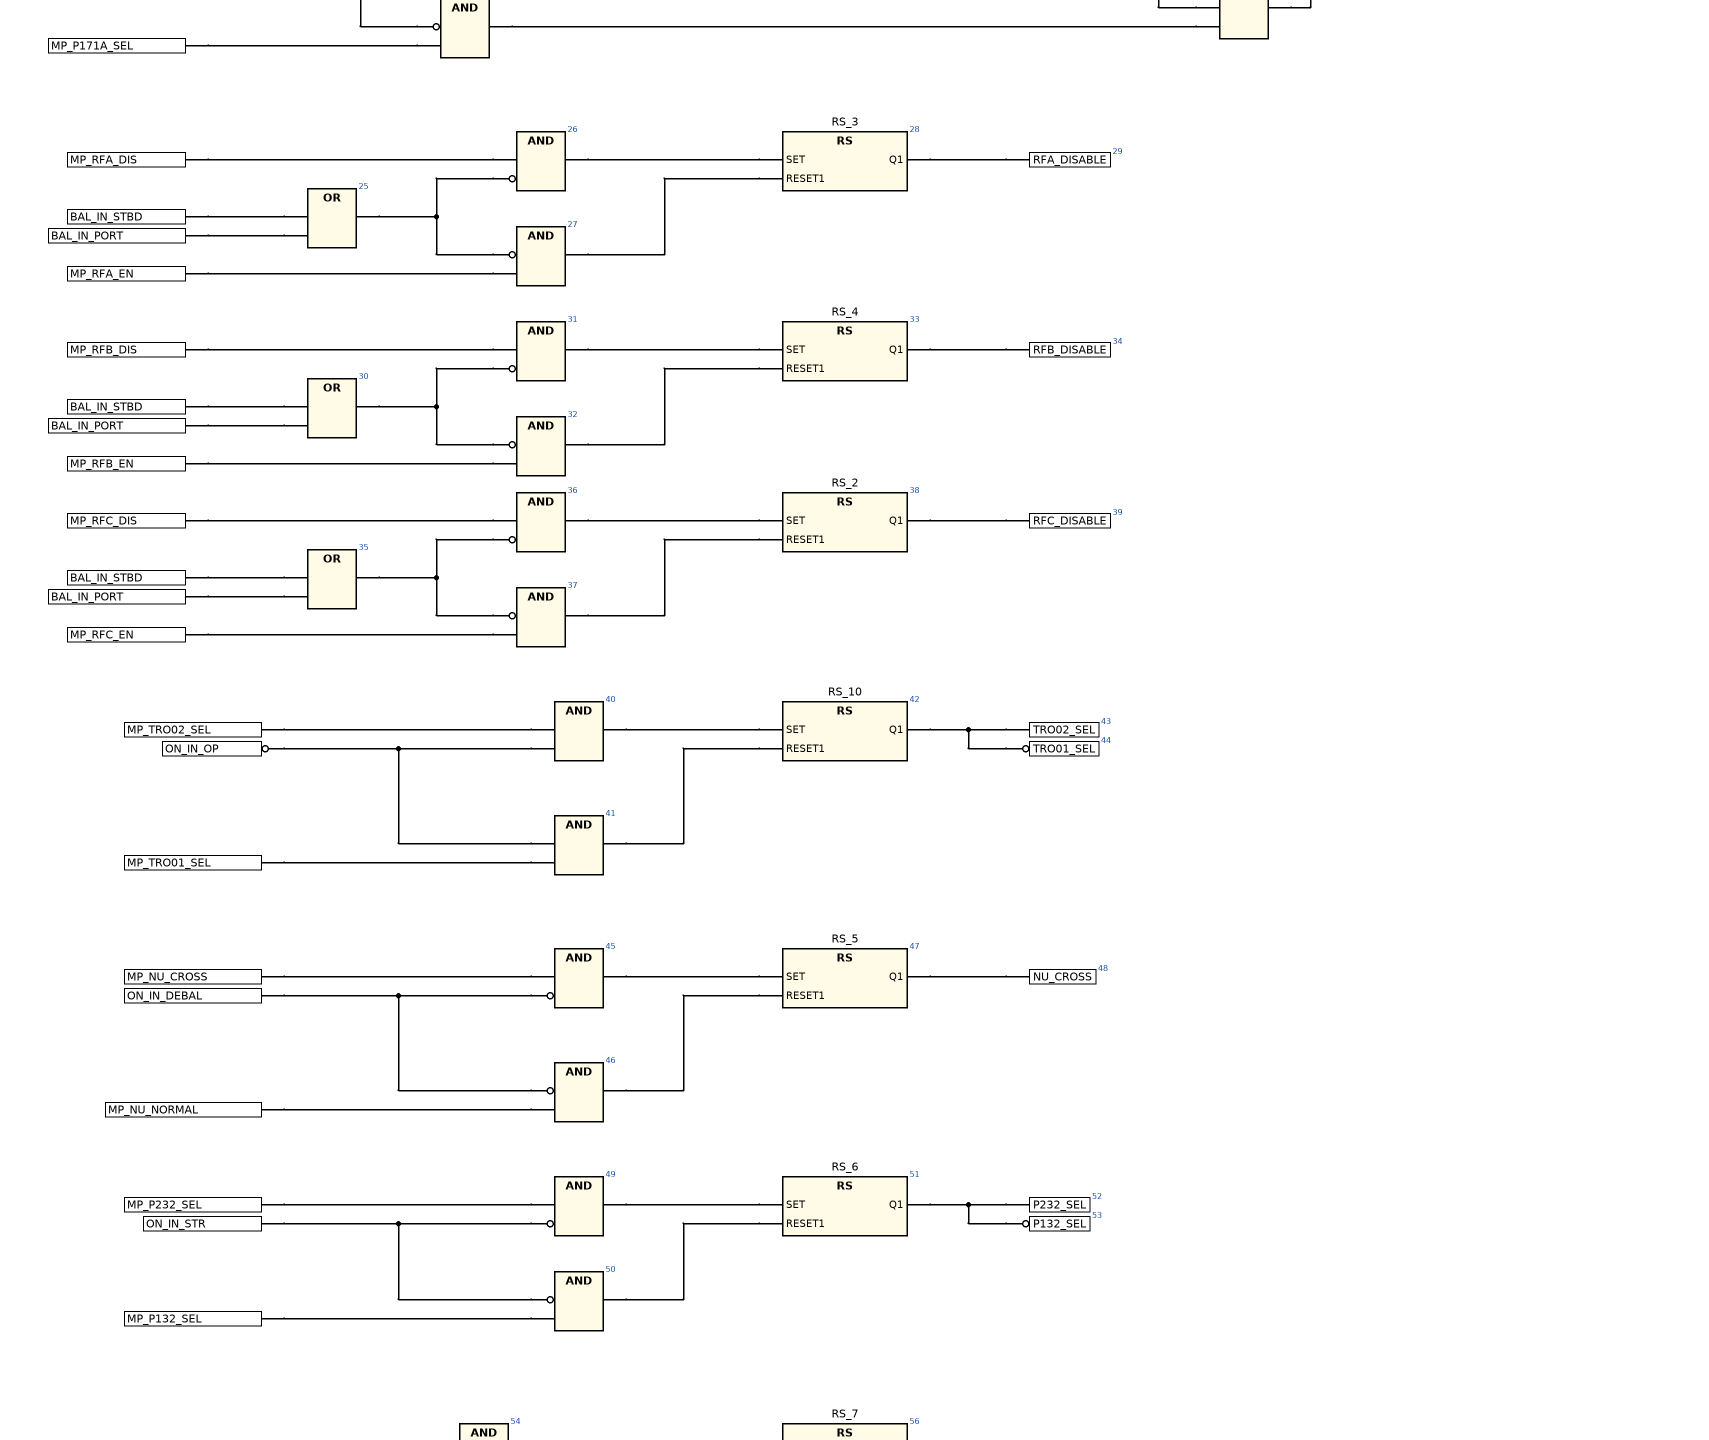
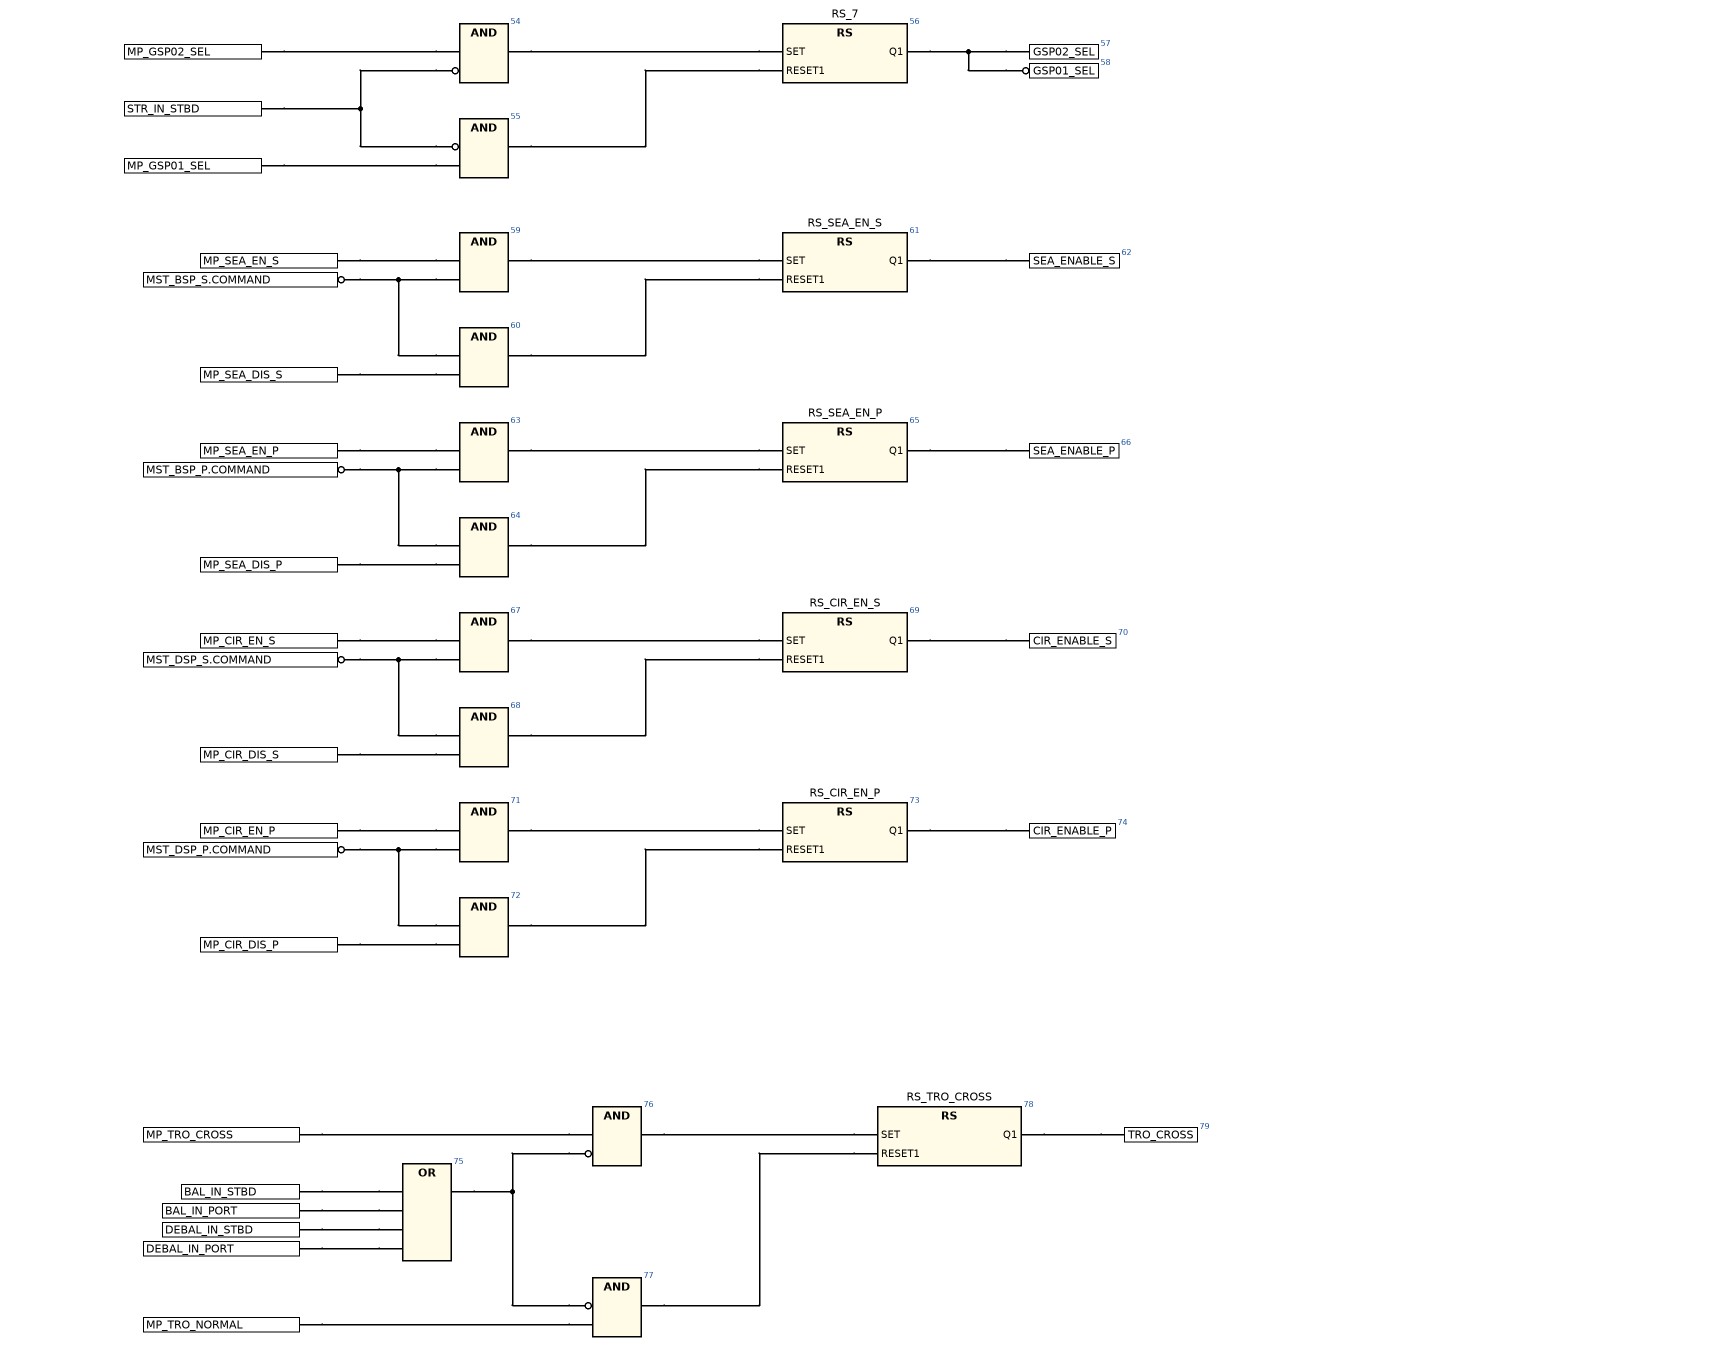
_w1 := ON_IN_BAL OR BLOWER_TIMER.BLR_GAS_SET.Q1;
RS_0(SET := MP_B117B_SEL AND NOT ON_IN_BAL OR B117A_SEL AND (B117A_STF OR XV1171A_OPF OR B_117A_F OR B_117A_OFF) AND _w1, RESET1 := NOT ON_IN_BAL AND MP_B117A_SEL OR _w1 AND B117B_SEL AND (B117B_STF OR XV1171B_OPF OR B_117B_F OR B_117B_OFF)); // RS
B117A_SEL := NOT RS_0.Q1;
B117B_SEL := RS_0.Q1;
_w2 := BAL_IN_STBD OR BAL_IN_PORT;
_w3 := BST_S_06.COMMAND OR BST_S_06.COMPLETE OR BST_P_06.COMMAND OR BST_P_06.COMPLETE;
RS_1(SET := MP_P171B_SEL AND NOT _w2 OR P171A_SEL AND (P171A_STF OR P_171A_OFF OR P_171A_F) AND _w3, RESET1 := _w3 AND P171B_SEL AND (P171B_STF OR P_171B_OFF OR P_171B_F) OR NOT _w2 AND MP_P171A_SEL); // RS
P171A_SEL := NOT RS_1.Q1;
P171B_SEL := RS_1.Q1;
_w4 := BAL_IN_STBD OR BAL_IN_PORT;
RS_3(SET := MP_RFA_DIS AND NOT _w4, RESET1 := NOT _w4 AND MP_RFA_EN); // RS
RFA_DISABLE := RS_3.Q1;
_w5 := BAL_IN_STBD OR BAL_IN_PORT;
RS_4(SET := MP_RFB_DIS AND NOT _w5, RESET1 := NOT _w5 AND MP_RFB_EN); // RS
RFB_DISABLE := RS_4.Q1;
_w6 := BAL_IN_STBD OR BAL_IN_PORT;
RS_2(SET := MP_RFC_DIS AND NOT _w6, RESET1 := NOT _w6 AND MP_RFC_EN); // RS
RFC_DISABLE := RS_2.Q1;
RS_10(SET := MP_TRO02_SEL AND NOT ON_IN_OP, RESET1 := NOT ON_IN_OP AND MP_TRO01_SEL); // RS
TRO02_SEL := RS_10.Q1;
TRO01_SEL := NOT RS_10.Q1;
RS_5(SET := MP_NU_CROSS AND NOT ON_IN_DEBAL, RESET1 := NOT ON_IN_DEBAL AND MP_NU_NORMAL); // RS
NU_CROSS := RS_5.Q1;
RS_6(SET := MP_P232_SEL AND NOT ON_IN_STR, RESET1 := NOT ON_IN_STR AND MP_P132_SEL); // RS
P232_SEL := RS_6.Q1;
P132_SEL := NOT RS_6.Q1;
RS_7(SET := MP_GSP02_SEL AND NOT STR_IN_STBD, RESET1 := NOT STR_IN_STBD AND MP_GSP01_SEL); // RS
GSP02_SEL := RS_7.Q1;
GSP01_SEL := NOT RS_7.Q1;
RS_SEA_EN_S(SET := MP_SEA_EN_S AND NOT MST_BSP_S.COMMAND, RESET1 := NOT MST_BSP_S.COMMAND AND MP_SEA_DIS_S); // RS
SEA_ENABLE_S := RS_SEA_EN_S.Q1;
RS_SEA_EN_P(SET := MP_SEA_EN_P AND NOT MST_BSP_P.COMMAND, RESET1 := NOT MST_BSP_P.COMMAND AND MP_SEA_DIS_P); // RS
SEA_ENABLE_P := RS_SEA_EN_P.Q1;
RS_CIR_EN_S(SET := MP_CIR_EN_S AND NOT MST_DSP_S.COMMAND, RESET1 := NOT MST_DSP_S.COMMAND AND MP_CIR_DIS_S); // RS
CIR_ENABLE_S := RS_CIR_EN_S.Q1;
RS_CIR_EN_P(SET := MP_CIR_EN_P AND NOT MST_DSP_P.COMMAND, RESET1 := NOT MST_DSP_P.COMMAND AND MP_CIR_DIS_P); // RS
CIR_ENABLE_P := RS_CIR_EN_P.Q1;
_w7 := BAL_IN_STBD OR BAL_IN_PORT OR DEBAL_IN_STBD OR DEBAL_IN_PORT;
RS_TRO_CROSS(SET := MP_TRO_CROSS AND NOT _w7, RESET1 := NOT _w7 AND MP_TRO_NORMAL); // RS
TRO_CROSS := RS_TRO_CROSS.Q1;

END_PROGRAM

// Device/Application/Logic/0.ETC/UTILITY
PROGRAM UTILITY
VAR
	INJECTION_SET: BWTS.INJECTION_SET;
	
		
	RS_BAL_ST_M : RS;
	TP_BAL_SP_M : TP;
	RS_DEBAL_ST_M : RS;
	TP_DEBAL_SP_M : TP;	
	RS_STRIP_ST : RS;
	TP_STRIP_SP : TP;
	
	RS_RFA_ST : RS;
	TP_RFA_SP : TP;
	RS_RFB_ST : RS;
	TP_RFB_SP : TP;
	RS_RFC_ST : RS;
	TP_RFC_SP : TP; 
	
	NA_PRE_SET_P132 : BWTS.NA_PRE_SET;
	NA_PRE_SET_P232 : BWTS.NA_PRE_SET;
		
	NA_CAPA_N1 : REAL := 31.2;
	NA_CAPA_N2 : REAL := 61.5;
	NA_CAPA_N3 : REAL := 129;
	NA_CAPA_N4 : REAL := 244.8;
END_VAR
VAR // added by the converter: edge detectors and wires of the graphical bodies
    _w1 : ANY;
END_VAR

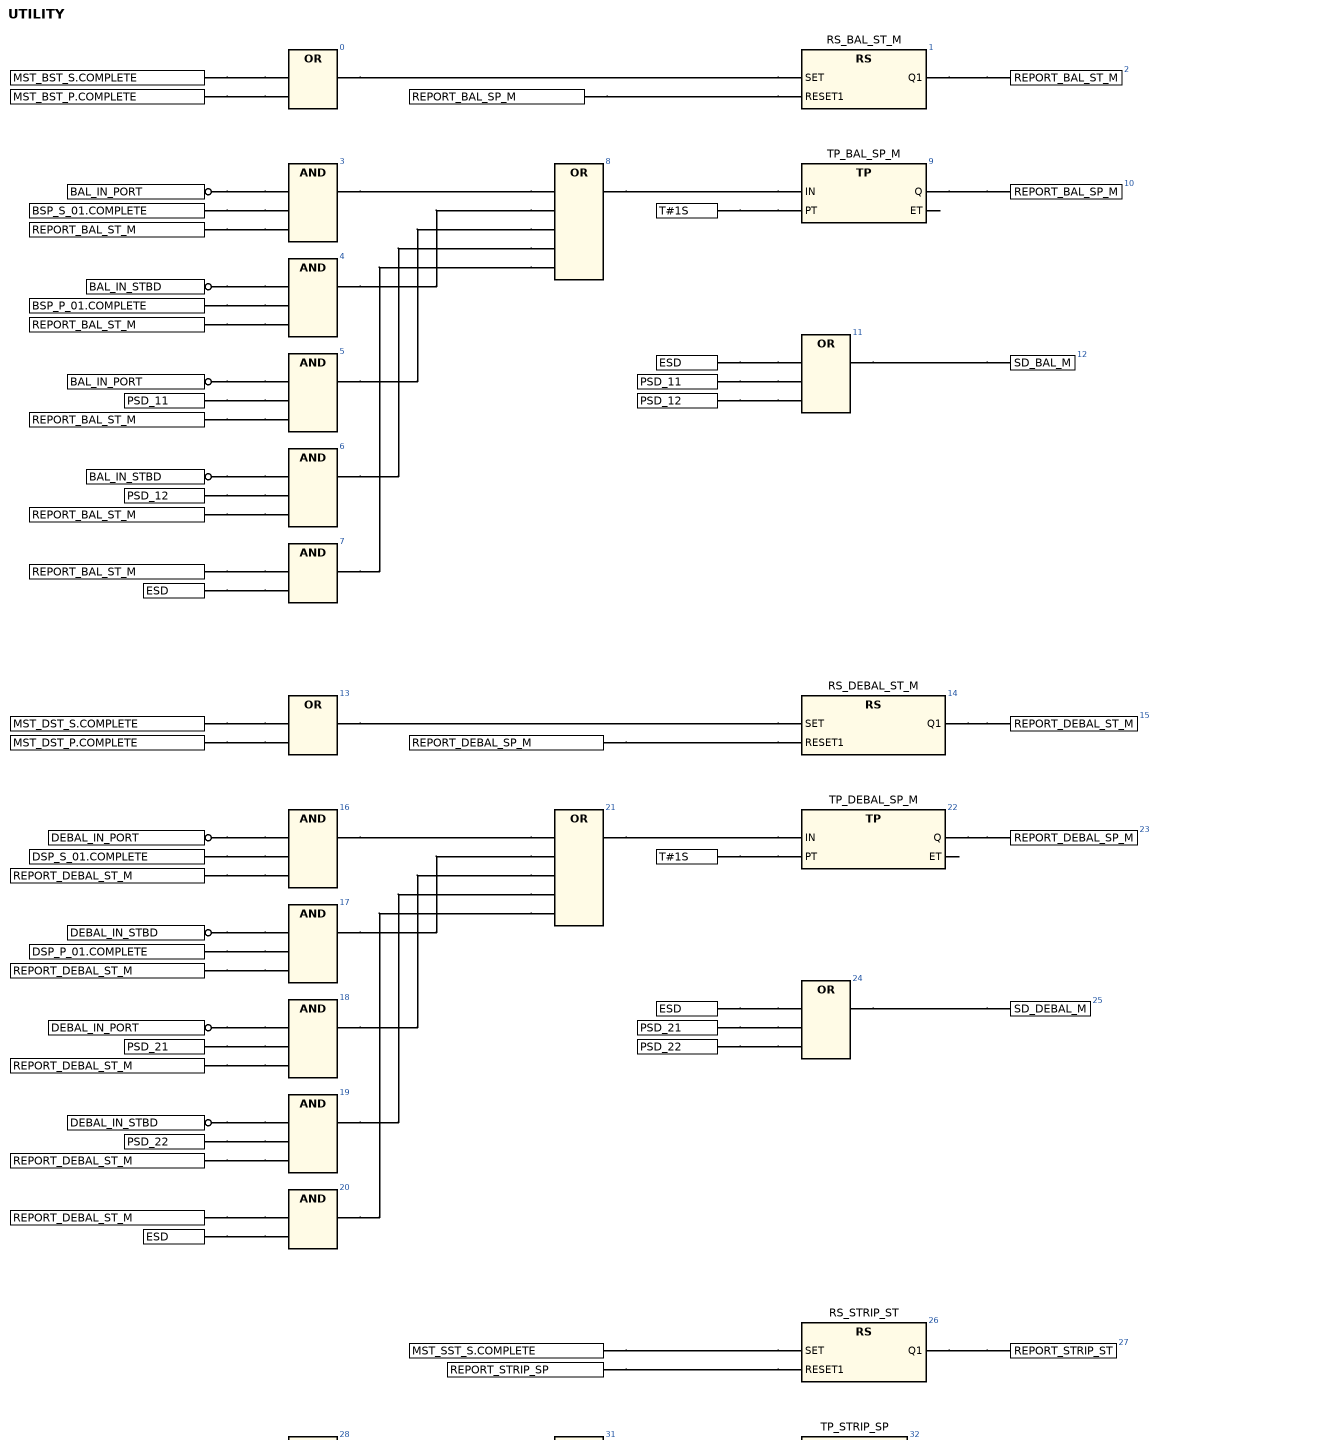
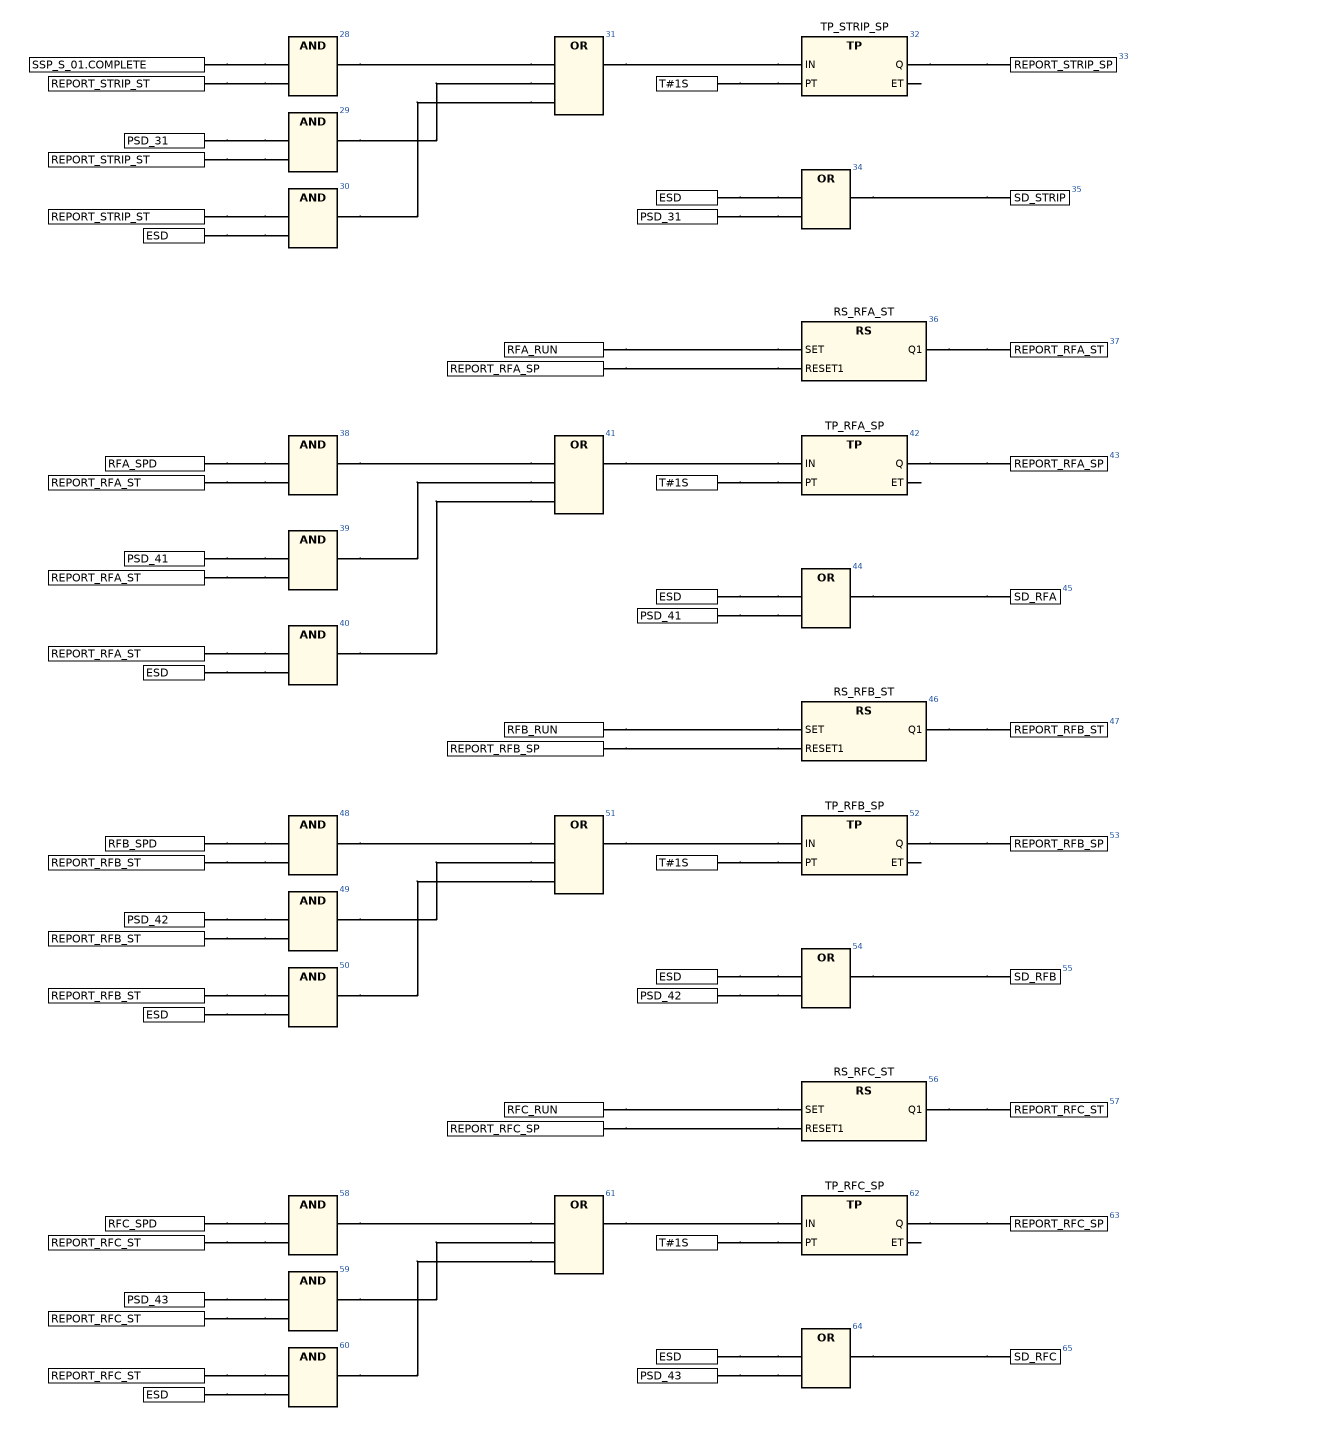
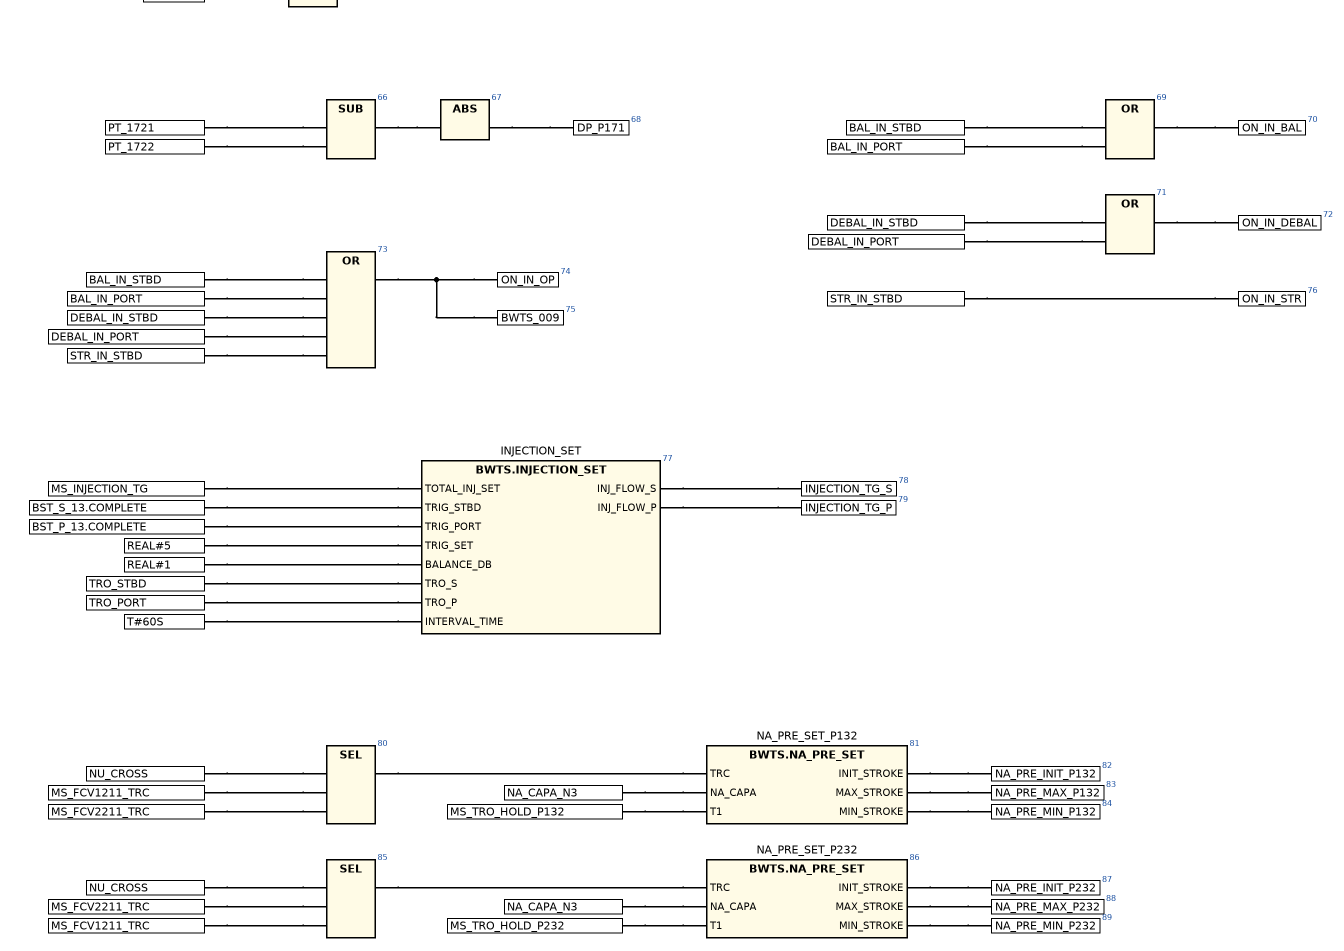
RS_BAL_ST_M(SET := MST_BST_S.COMPLETE OR MST_BST_P.COMPLETE, RESET1 := REPORT_BAL_SP_M); // RS
REPORT_BAL_ST_M := RS_BAL_ST_M.Q1;
TP_BAL_SP_M(IN := NOT BAL_IN_PORT AND BSP_S_01.COMPLETE AND REPORT_BAL_ST_M OR NOT BAL_IN_STBD AND BSP_P_01.COMPLETE AND REPORT_BAL_ST_M OR NOT BAL_IN_PORT AND PSD_11 AND REPORT_BAL_ST_M OR NOT BAL_IN_STBD AND PSD_12 AND REPORT_BAL_ST_M OR REPORT_BAL_ST_M AND ESD, PT := T#1S); // TP
REPORT_BAL_SP_M := TP_BAL_SP_M.Q;
SD_BAL_M := ESD OR PSD_11 OR PSD_12;
RS_DEBAL_ST_M(SET := MST_DST_S.COMPLETE OR MST_DST_P.COMPLETE, RESET1 := REPORT_DEBAL_SP_M); // RS
REPORT_DEBAL_ST_M := RS_DEBAL_ST_M.Q1;
TP_DEBAL_SP_M(IN := NOT DEBAL_IN_PORT AND DSP_S_01.COMPLETE AND REPORT_DEBAL_ST_M OR NOT DEBAL_IN_STBD AND DSP_P_01.COMPLETE AND REPORT_DEBAL_ST_M OR NOT DEBAL_IN_PORT AND PSD_21 AND REPORT_DEBAL_ST_M OR NOT DEBAL_IN_STBD AND PSD_22 AND REPORT_DEBAL_ST_M OR REPORT_DEBAL_ST_M AND ESD, PT := T#1S); // TP
REPORT_DEBAL_SP_M := TP_DEBAL_SP_M.Q;
SD_DEBAL_M := ESD OR PSD_21 OR PSD_22;
RS_STRIP_ST(SET := MST_SST_S.COMPLETE, RESET1 := REPORT_STRIP_SP); // RS
REPORT_STRIP_ST := RS_STRIP_ST.Q1;
TP_STRIP_SP(IN := SSP_S_01.COMPLETE AND REPORT_STRIP_ST OR PSD_31 AND REPORT_STRIP_ST OR REPORT_STRIP_ST AND ESD, PT := T#1S); // TP
REPORT_STRIP_SP := TP_STRIP_SP.Q;
SD_STRIP := ESD OR PSD_31;
RS_RFA_ST(SET := RFA_RUN, RESET1 := REPORT_RFA_SP); // RS
REPORT_RFA_ST := RS_RFA_ST.Q1;
TP_RFA_SP(IN := RFA_SPD AND REPORT_RFA_ST OR PSD_41 AND REPORT_RFA_ST OR REPORT_RFA_ST AND ESD, PT := T#1S); // TP
REPORT_RFA_SP := TP_RFA_SP.Q;
SD_RFA := ESD OR PSD_41;
RS_RFB_ST(SET := RFB_RUN, RESET1 := REPORT_RFB_SP); // RS
REPORT_RFB_ST := RS_RFB_ST.Q1;
TP_RFB_SP(IN := RFB_SPD AND REPORT_RFB_ST OR PSD_42 AND REPORT_RFB_ST OR REPORT_RFB_ST AND ESD, PT := T#1S); // TP
REPORT_RFB_SP := TP_RFB_SP.Q;
SD_RFB := ESD OR PSD_42;
RS_RFC_ST(SET := RFC_RUN, RESET1 := REPORT_RFC_SP); // RS
REPORT_RFC_ST := RS_RFC_ST.Q1;
TP_RFC_SP(IN := RFC_SPD AND REPORT_RFC_ST OR PSD_43 AND REPORT_RFC_ST OR REPORT_RFC_ST AND ESD, PT := T#1S); // TP
REPORT_RFC_SP := TP_RFC_SP.Q;
SD_RFC := ESD OR PSD_43;
DP_P171 := ABS(PT_1721 - PT_1722);
ON_IN_BAL := BAL_IN_STBD OR BAL_IN_PORT;
ON_IN_DEBAL := DEBAL_IN_STBD OR DEBAL_IN_PORT;
_w1 := BAL_IN_STBD OR BAL_IN_PORT OR DEBAL_IN_STBD OR DEBAL_IN_PORT OR STR_IN_STBD;
ON_IN_OP := _w1;
BWTS_009 := _w1;
ON_IN_STR := STR_IN_STBD;
INJECTION_SET(
    TOTAL_INJ_SET := MS_INJECTION_TG,
    TRIG_STBD := BST_S_13.COMPLETE,
    TRIG_PORT := BST_P_13.COMPLETE,
    TRIG_SET := REAL#5,
    BALANCE_DB := REAL#1,
    TRO_S := TRO_STBD,
    TRO_P := TRO_PORT,
    INTERVAL_TIME := T#60S); // BWTS.INJECTION_SET
INJECTION_TG_S := INJECTION_SET.INJ_FLOW_S;
INJECTION_TG_P := INJECTION_SET.INJ_FLOW_P;
NA_PRE_SET_P132(
    TRC := SEL(NU_CROSS, MS_FCV1211_TRC, MS_FCV2211_TRC),
    NA_CAPA := NA_CAPA_N3,
    T1 := MS_TRO_HOLD_P132); // BWTS.NA_PRE_SET
NA_PRE_INIT_P132 := NA_PRE_SET_P132.INIT_STROKE;
NA_PRE_MAX_P132 := NA_PRE_SET_P132.MAX_STROKE;
NA_PRE_MIN_P132 := NA_PRE_SET_P132.MIN_STROKE;
NA_PRE_SET_P232(
    TRC := SEL(NU_CROSS, MS_FCV2211_TRC, MS_FCV1211_TRC),
    NA_CAPA := NA_CAPA_N3,
    T1 := MS_TRO_HOLD_P232); // BWTS.NA_PRE_SET
NA_PRE_INIT_P232 := NA_PRE_SET_P232.INIT_STROKE;
NA_PRE_MAX_P232 := NA_PRE_SET_P232.MAX_STROKE;
NA_PRE_MIN_P232 := NA_PRE_SET_P232.MIN_STROKE;

END_PROGRAM

// Device/Application/Logic/0.ETC/RUNNING_HOURS
PROGRAM RUNNING_HOURS
VAR
	RH_ELECT_TOTAL, RH_ELECT_PARTIAL: BWTS.RH_100MS;
	
	RH_AIT1121, RH_AIT1122, RH_AIT1123: BWTS.RH_100MS;
	
	RH_P171A, RH_P171B: BWTS.RH_100MS;
	
	RH_P132, RH_P232: BWTS.RH_100MS;
	
	RH_AIT151, RH_AIT251: BWTS.RH_100MS;
	
	RH_BAL_M : BWTS.RH_100MS;
	RH_DEBAL_M : BWTS.RH_100MS;
	RH_STRIP : BWTS.RH_100MS;
END_VAR

////////////////////////////////////////////////////////////////// FOR PERIOD MAINTENANCE////////////////////////////////////////////////////////////////// 
// ELECTROLYZER TOTAL/PARTIAL RUNNING HOUR
RH_ELECT_TOTAL(bTrigger := RFA_RUN OR RFB_RUN OR RFC_RUN, bReset := MP_RH_EM_TOTAL_RESET, udTimer := TIME_RH_EM_TOTAL, udTimeToHour =>TIME_TOTAL_HOUR_EM_TOTAL);
RH_ELECT_PARTIAL(bTrigger := RFA_RUN OR RFB_RUN OR RFC_RUN, bReset := MP_RH_EM_PARTIAL_RESET, udTimer := TIME_RH_EM_PARTIAL, udTimeToHour =>TIME_TOTAL_HOUR_EM_PARTIAL);

// H2 GAS DETECTOR(AIT-1121/1122/1123) RUNNING HOUR
RH_AIT1121(bTrigger := TRUE, bReset := MP_RH_AIT1121_RESET, udTimer := TIME_RH_AIT1121, udDay =>TIME_TOTAL_DAY_AIT1121);
RH_AIT1122(bTrigger := TRUE, bReset := MP_RH_AIT1122_RESET, udTimer := TIME_RH_AIT1122, udDay =>TIME_TOTAL_DAY_AIT1122);
RH_AIT1123(bTrigger := TRUE, bReset := MP_RH_AIT1123_RESET, udTimer := TIME_RH_AIT1123, udDay =>TIME_TOTAL_DAY_AIT1123);

// SEA WATER FEED PUMP(P-171A/B) RUNNING HOUR
RH_P171A(bTrigger := TRUE, bReset := MP_RH_P171A_RESET, udTimer := TIME_RH_P171A, udDay =>TIME_TOTAL_DAY_P171A); 
RH_P171B(bTrigger := TRUE, bReset := MP_RH_P171B_RESET, udTimer := TIME_RH_P171B, udDay =>TIME_TOTAL_DAY_P171B);

// N.A PUMP(P-132/232/332) RUNNING HOUR
RH_P132(bTrigger := P132_RUN, bReset := MP_RH_P132_RESET, udTimer := TIME_RH_P132, udTimeToHour =>TIME_TOTAL_HOUR_P132);
RH_P232(bTrigger := P232_RUN, bReset := MP_RH_P232_RESET, udTimer := TIME_RH_P232, udTimeToHour =>TIME_TOTAL_HOUR_P232);

// TRO(AIT-151/251/351) RUNNING HOUR
RH_AIT151(bTrigger := TRUE, bReset := MP_RH_AIT151_RESET, udTimer := TIME_RH_AIT151, udDay =>TIME_TOTAL_DAY_AIT151);
RH_AIT251(bTrigger := TRUE, bReset := MP_RH_AIT251_RESET, udTimer := TIME_RH_AIT251, udDay =>TIME_TOTAL_DAY_AIT251);

////////////////////////////////////////////////////////////////// FOR OPERATION RUNNING TIME //////////////////////////////////////////////////////////////////
// MAIN BALLASTING OPERATION RUNNING HOUR
RH_BAL_M(bTrigger := REPORT_BAL_ST_M, bReset := MP_RH_BAL_M_RESET, udTimer := TIME_RH_BAL_M, udDay => TIME_DAY_RH_BAL_M, udHour => TIME_HOUR_RH_BAL_M, udMin => TIME_MIN_RH_BAL_M);

// MAIN DEBALLASTING OPERATION RUNNING HOUR
RH_DEBAL_M(bTrigger := REPORT_DEBAL_ST_M, bReset := MP_RH_DEBAL_M_RESET, udTimer := TIME_RH_DEBAL_M, udDay => TIME_DAY_RH_DEBAL_M, udHour => TIME_HOUR_RH_DEBAL_M, udMin => TIME_MIN_RH_DEBAL_M);

// APT DEBALLASTING OPERATION RUNNING HOUR
RH_STRIP(bTrigger := REPORT_STRIP_ST, bReset := MP_RH_STRIP_RESET, udTimer := TIME_RH_STRIP, udDay => TIME_DAY_RH_STRIP, udHour => TIME_HOUR_RH_STRIP, udMin => TIME_MIN_RH_STRIP);

END_PROGRAM

// Device/Application/Logic/4.Device/DEVICE_AIT151
PROGRAM DEVICE_AIT151
VAR
	AIT151: BWTS.DEVICE;
END_VAR
VAR // added by the converter: edge detectors and wires of the graphical bodies
    _w1, _w2, _w3, _w4, _w5, _w6 : BOOL;
    _w7, _w8, _w9 : ANY;
END_VAR

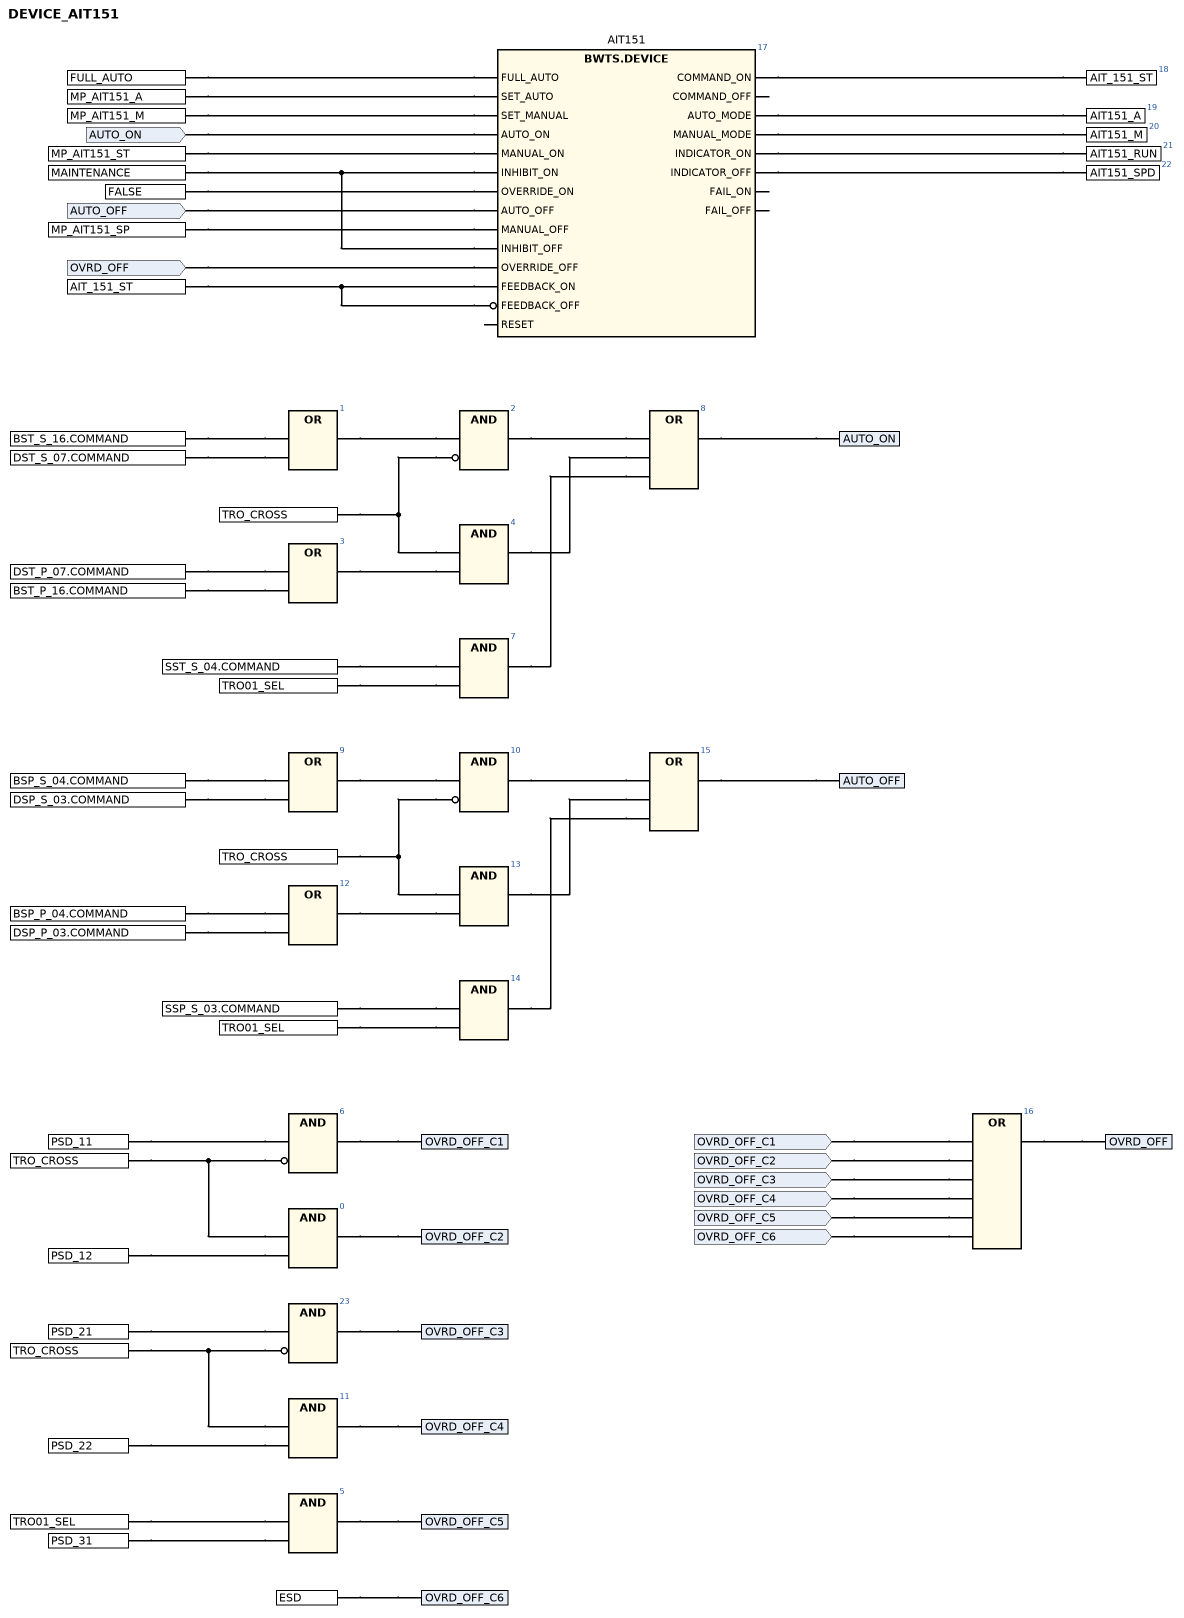
(* TRO_CROSS AND PSD_12; result not used *)
(* TRO01_SEL AND PSD_31; result not used *)
(* PSD_11 AND NOT TRO_CROSS; result not used *)
(* (BST_S_16.COMMAND OR DST_S_07.COMMAND) AND NOT TRO_CROSS OR TRO_CROSS AND (DST_P_07.COMMAND OR BST_P_16.COMMAND) OR SST_S_04.COMMAND AND TRO01_SEL; result not used *)
(* TRO_CROSS AND PSD_22; result not used *)
(* (BSP_S_04.COMMAND OR DSP_S_03.COMMAND) AND NOT TRO_CROSS OR TRO_CROSS AND (BSP_P_04.COMMAND OR DSP_P_03.COMMAND) OR SSP_S_03.COMMAND AND TRO01_SEL; result not used *)
(* _w1 OR _w2 OR _w3 OR _w4 OR _w5 OR _w6; result not used *)
AIT151(
    FULL_AUTO := FULL_AUTO,
    SET_AUTO := MP_AIT151_A,
    SET_MANUAL := MP_AIT151_M,
    AUTO_ON := _w7,
    MANUAL_ON := MP_AIT151_ST,
    INHIBIT_ON := MAINTENANCE,
    OVERRIDE_ON := FALSE,
    AUTO_OFF := _w8,
    MANUAL_OFF := MP_AIT151_SP,
    INHIBIT_OFF := MAINTENANCE,
    OVERRIDE_OFF := _w9,
    FEEDBACK_ON := AIT_151_ST,
    FEEDBACK_OFF := NOT AIT_151_ST); // BWTS.DEVICE
AIT_151_ST := AIT151.COMMAND_ON;
AIT151_A := AIT151.AUTO_MODE;
AIT151_M := AIT151.MANUAL_MODE;
AIT151_RUN := AIT151.INDICATOR_ON;
AIT151_SPD := AIT151.INDICATOR_OFF;
(* PSD_21 AND NOT TRO_CROSS; result not used *)

END_PROGRAM

// Device/Application/Logic/4.Device/DEVICE_AIT251
PROGRAM DEVICE_AIT251
VAR
	AIT251: BWTS.DEVICE;
END_VAR
VAR // added by the converter: edge detectors and wires of the graphical bodies
    _w1, _w2, _w3, _w4, _w5, _w6 : BOOL;
    _w7, _w8, _w9 : ANY;
END_VAR

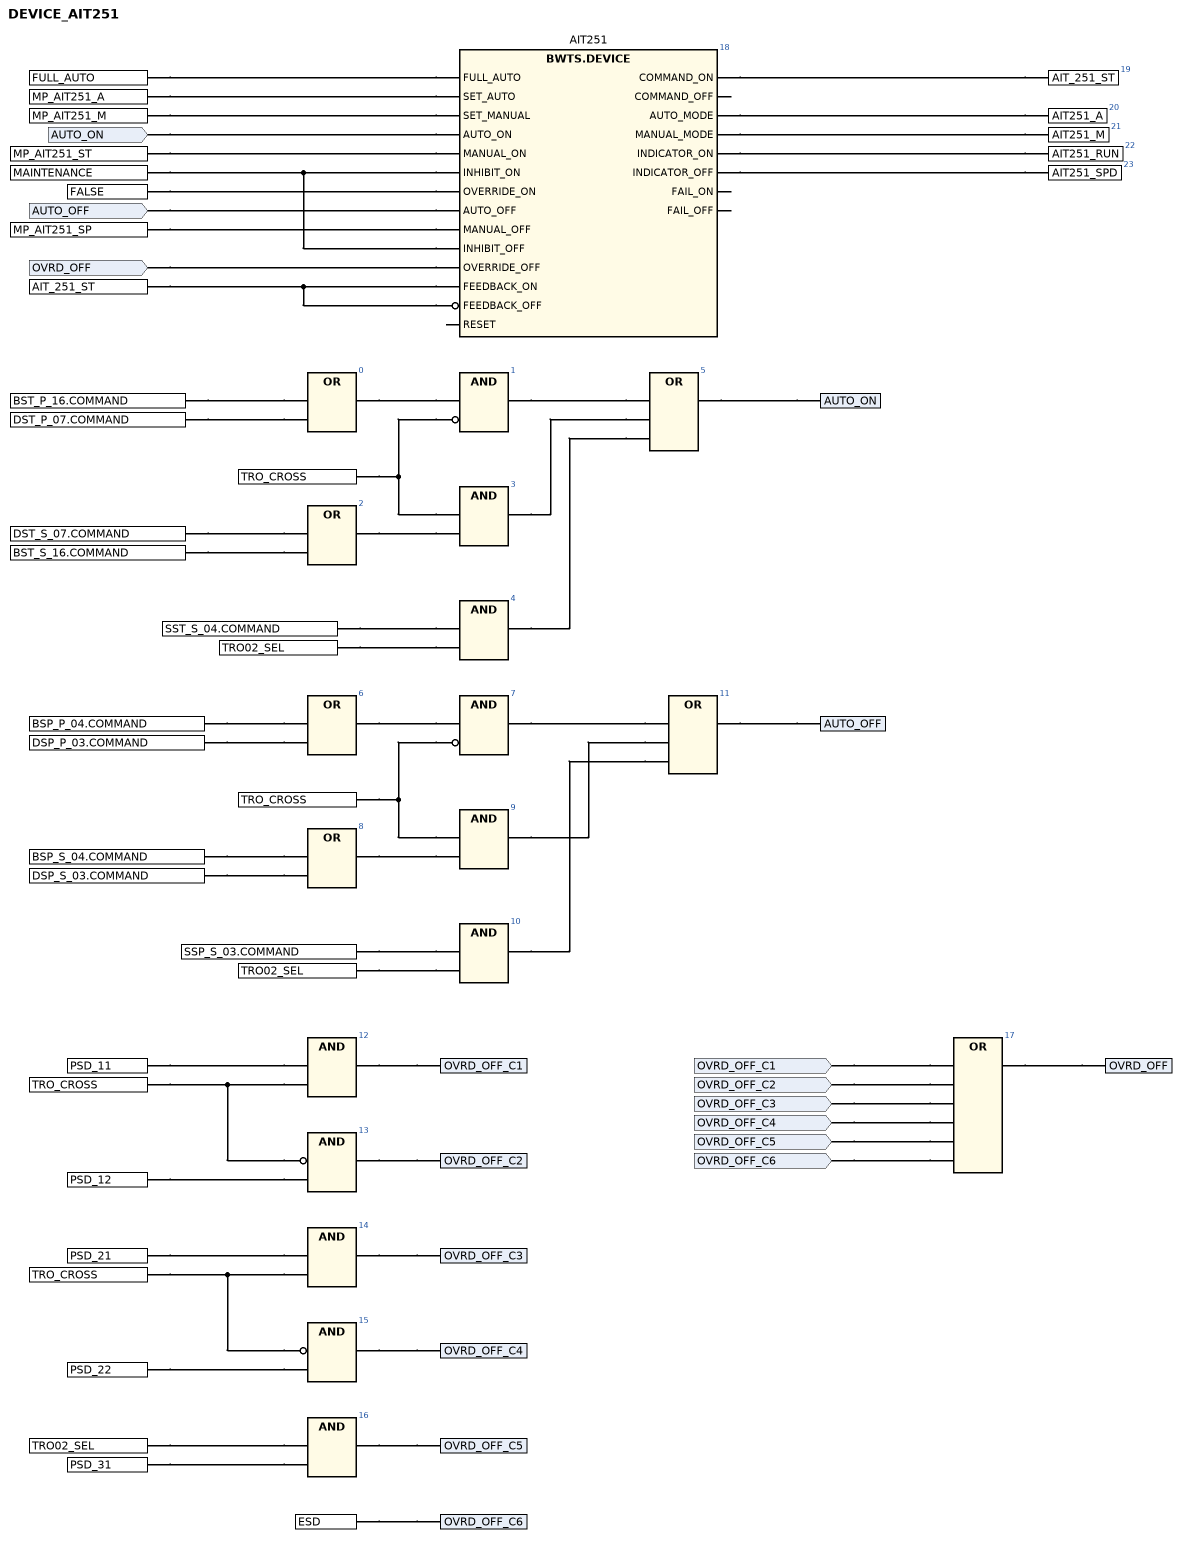
(* (BST_P_16.COMMAND OR DST_P_07.COMMAND) AND NOT TRO_CROSS OR TRO_CROSS AND (DST_S_07.COMMAND OR BST_S_16.COMMAND) OR SST_S_04.COMMAND AND TRO02_SEL; result not used *)
(* (BSP_P_04.COMMAND OR DSP_P_03.COMMAND) AND NOT TRO_CROSS OR TRO_CROSS AND (BSP_S_04.COMMAND OR DSP_S_03.COMMAND) OR SSP_S_03.COMMAND AND TRO02_SEL; result not used *)
(* PSD_11 AND TRO_CROSS; result not used *)
(* NOT TRO_CROSS AND PSD_12; result not used *)
(* PSD_21 AND TRO_CROSS; result not used *)
(* NOT TRO_CROSS AND PSD_22; result not used *)
(* TRO02_SEL AND PSD_31; result not used *)
(* _w1 OR _w2 OR _w3 OR _w4 OR _w5 OR _w6; result not used *)
AIT251(
    FULL_AUTO := FULL_AUTO,
    SET_AUTO := MP_AIT251_A,
    SET_MANUAL := MP_AIT251_M,
    AUTO_ON := _w7,
    MANUAL_ON := MP_AIT251_ST,
    INHIBIT_ON := MAINTENANCE,
    OVERRIDE_ON := FALSE,
    AUTO_OFF := _w8,
    MANUAL_OFF := MP_AIT251_SP,
    INHIBIT_OFF := MAINTENANCE,
    OVERRIDE_OFF := _w9,
    FEEDBACK_ON := AIT_251_ST,
    FEEDBACK_OFF := NOT AIT_251_ST); // BWTS.DEVICE
AIT_251_ST := AIT251.COMMAND_ON;
AIT251_A := AIT251.AUTO_MODE;
AIT251_M := AIT251.MANUAL_MODE;
AIT251_RUN := AIT251.INDICATOR_ON;
AIT251_SPD := AIT251.INDICATOR_OFF;

END_PROGRAM

// Device/Application/Logic/4.Device/DEVICE_GSP01
PROGRAM DEVICE_GSP01
VAR
TP_0: TP;
END_VAR
VAR // added by the converter: edge detectors and wires of the graphical bodies
    _w1 : ANY;
END_VAR

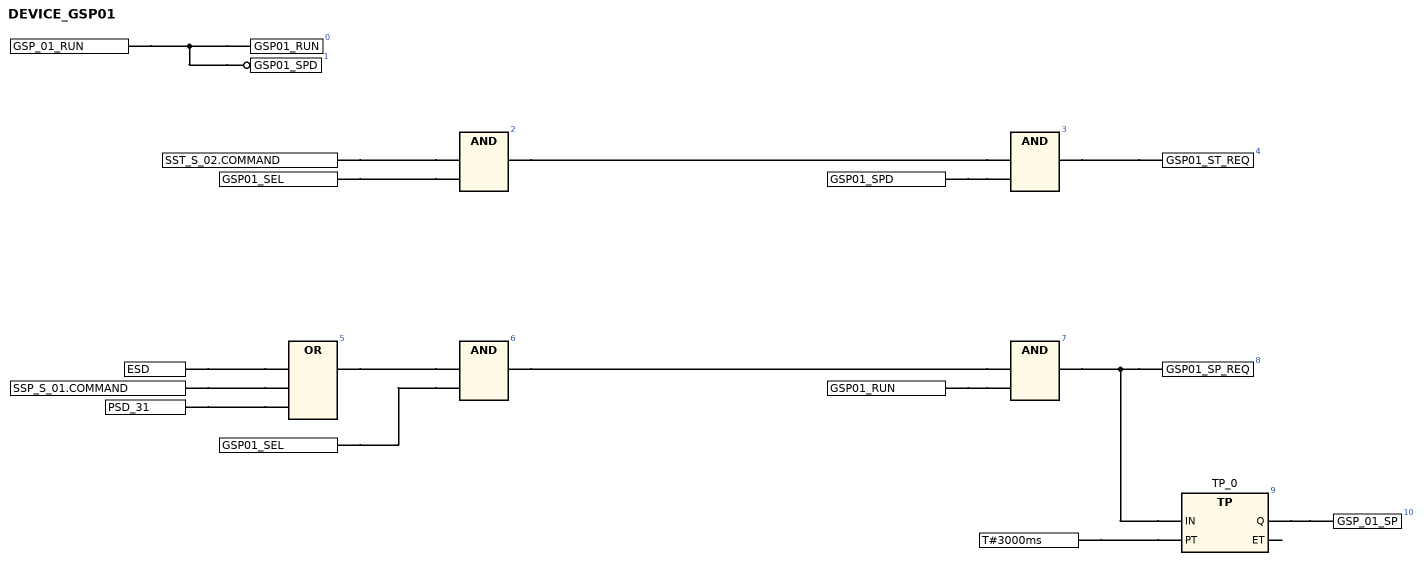
GSP01_RUN := GSP_01_RUN;
GSP01_SPD := NOT GSP_01_RUN;
GSP01_ST_REQ := (SST_S_02.COMMAND AND GSP01_SEL) AND GSP01_SPD;
_w1 := ((ESD OR SSP_S_01.COMMAND OR PSD_31) AND GSP01_SEL) AND GSP01_RUN;
GSP01_SP_REQ := _w1;
TP_0(IN := _w1, PT := T#3000ms); // TP
GSP_01_SP := TP_0.Q;

END_PROGRAM

// Device/Application/Logic/4.Device/DEVICE_GSP02
PROGRAM DEVICE_GSP02
VAR
TP_0: TP;
END_VAR
VAR // added by the converter: edge detectors and wires of the graphical bodies
    _w1 : ANY;
END_VAR

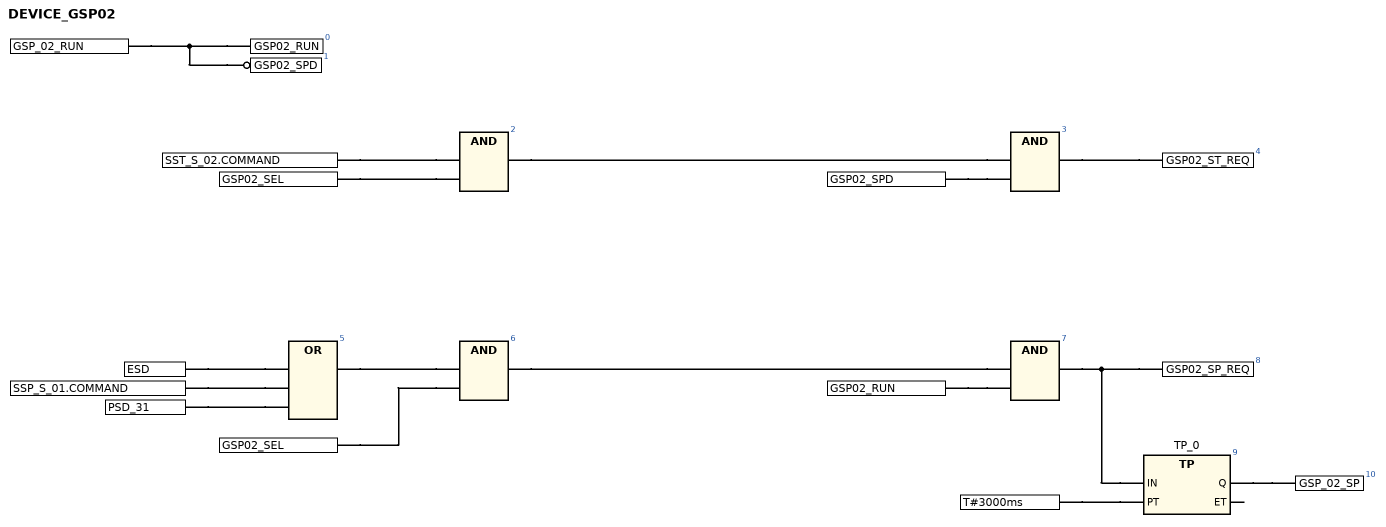
GSP02_RUN := GSP_02_RUN;
GSP02_SPD := NOT GSP_02_RUN;
GSP02_ST_REQ := (SST_S_02.COMMAND AND GSP02_SEL) AND GSP02_SPD;
_w1 := ((ESD OR SSP_S_01.COMMAND OR PSD_31) AND GSP02_SEL) AND GSP02_RUN;
GSP02_SP_REQ := _w1;
TP_0(IN := _w1, PT := T#3000ms); // TP
GSP_02_SP := TP_0.Q;

END_PROGRAM

// Device/Application/Logic/4.Device/DEVICE_WBP01
PROGRAM DEVICE_WBP01
VAR

END_VAR

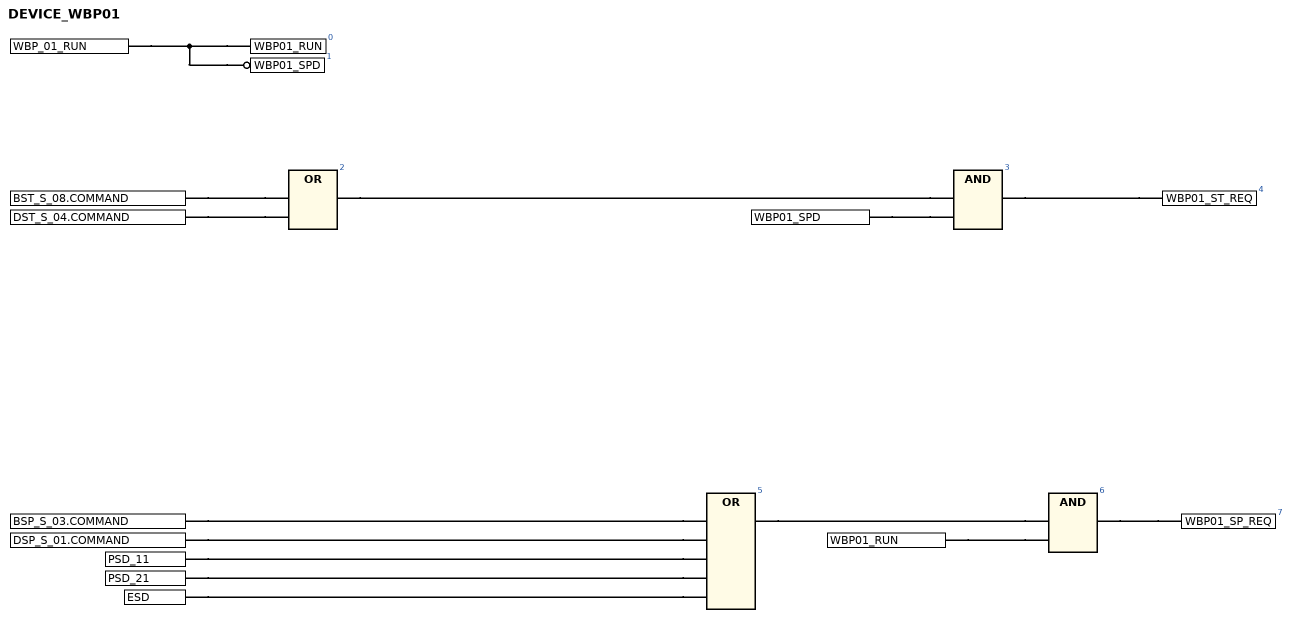
WBP01_RUN := WBP_01_RUN;
WBP01_SPD := NOT WBP_01_RUN;
WBP01_ST_REQ := (BST_S_08.COMMAND OR DST_S_04.COMMAND) AND WBP01_SPD;
WBP01_SP_REQ := (BSP_S_03.COMMAND OR DSP_S_01.COMMAND OR PSD_11 OR PSD_21 OR ESD) AND WBP01_RUN;

END_PROGRAM

// Device/Application/Logic/4.Device/DEVICE_WBP02
PROGRAM DEVICE_WBP02
VAR

END_VAR

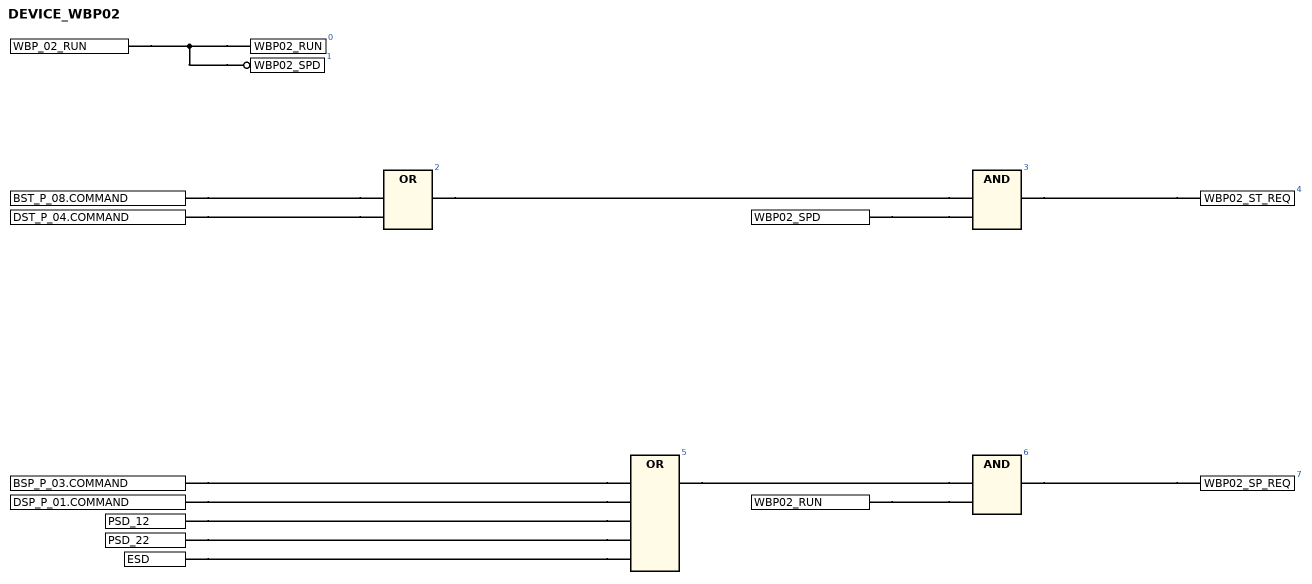
WBP02_RUN := WBP_02_RUN;
WBP02_SPD := NOT WBP_02_RUN;
WBP02_ST_REQ := (BST_P_08.COMMAND OR DST_P_04.COMMAND) AND WBP02_SPD;
WBP02_SP_REQ := (BSP_P_03.COMMAND OR DSP_P_01.COMMAND OR PSD_12 OR PSD_22 OR ESD) AND WBP02_RUN;

END_PROGRAM

// Device/Application/Logic/4.Device/DEVICE_XV1151
PROGRAM DEVICE_XV1151
VAR
	XV1151: BWTS.DEVICE;
	AUTO_ON : BOOL;
	AUTO_OFF : BOOL;
	OVRD_OFF : BOOL;
	
	TON_0: TON;
	TON_1: TON;
	TP_0: TP;	
END_VAR

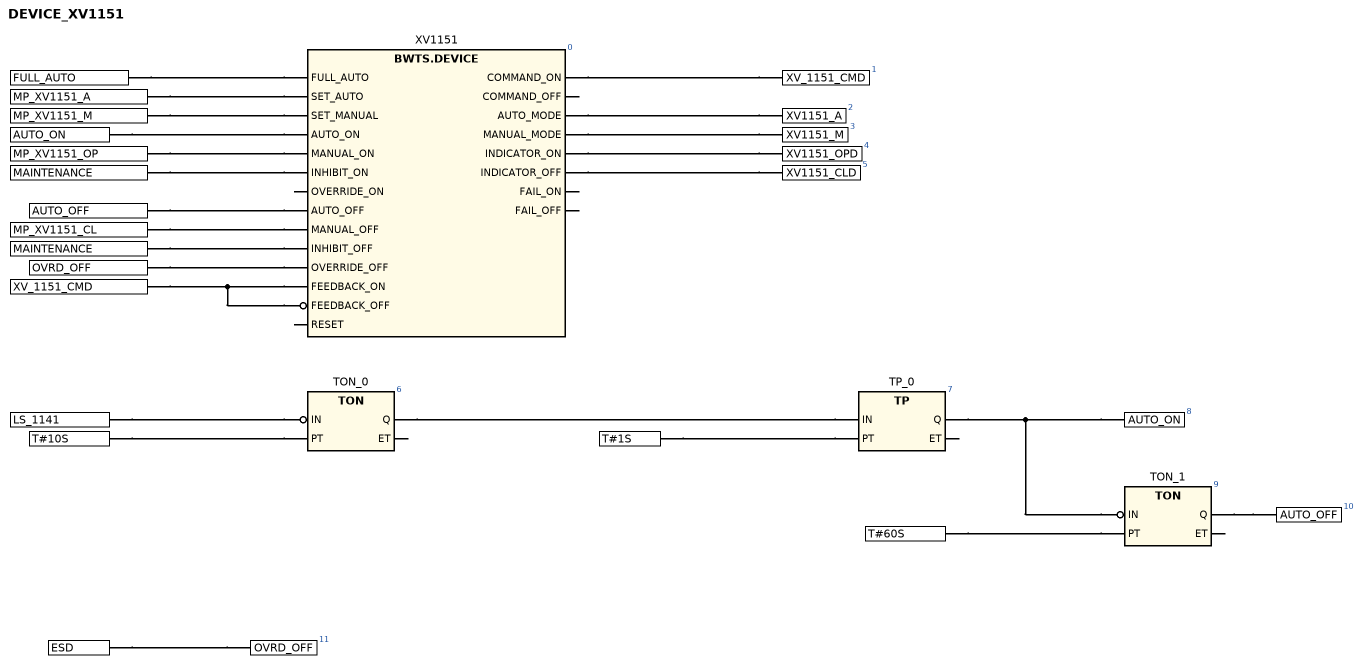
XV1151(
    FULL_AUTO := FULL_AUTO,
    SET_AUTO := MP_XV1151_A,
    SET_MANUAL := MP_XV1151_M,
    AUTO_ON := AUTO_ON,
    MANUAL_ON := MP_XV1151_OP,
    INHIBIT_ON := MAINTENANCE,
    AUTO_OFF := AUTO_OFF,
    MANUAL_OFF := MP_XV1151_CL,
    INHIBIT_OFF := MAINTENANCE,
    OVERRIDE_OFF := OVRD_OFF,
    FEEDBACK_ON := XV_1151_CMD,
    FEEDBACK_OFF := NOT XV_1151_CMD); // BWTS.DEVICE
XV_1151_CMD := XV1151.COMMAND_ON;
XV1151_A := XV1151.AUTO_MODE;
XV1151_M := XV1151.MANUAL_MODE;
XV1151_OPD := XV1151.INDICATOR_ON;
XV1151_CLD := XV1151.INDICATOR_OFF;
TON_0(IN := NOT LS_1141, PT := T#10S); // TON
TP_0(IN := TON_0.Q, PT := T#1S); // TP
AUTO_ON := TP_0.Q;
TON_1(IN := NOT TP_0.Q, PT := T#60S); // TON
AUTO_OFF := TON_1.Q;
OVRD_OFF := ESD;

END_PROGRAM

// Device/Application/Logic/4.Device/DEVICE_XV1172A
PROGRAM DEVICE_XV1172A
VAR
	TP_0: TP;
	RS_0: RS;
END_VAR
VAR // added by the converter: edge detectors and wires of the graphical bodies
    _w1, _w2 : ANY;
END_VAR

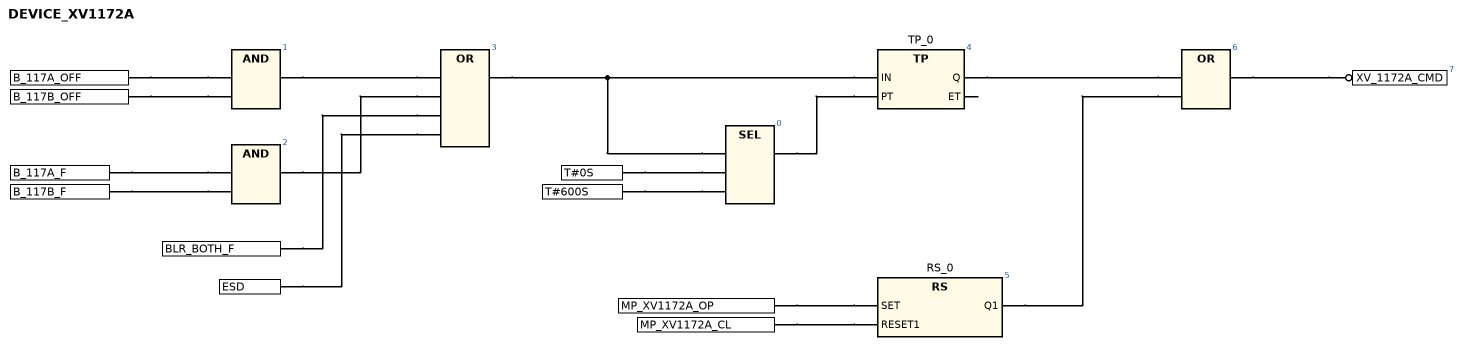
_w2 := SEL(_w1, T#0S, T#600S);
_w1 := B_117A_OFF AND B_117B_OFF OR B_117A_F AND B_117B_F OR BLR_BOTH_F OR ESD;
TP_0(IN := _w1, PT := _w2); // TP
RS_0(SET := MP_XV1172A_OP, RESET1 := MP_XV1172A_CL); // RS
XV_1172A_CMD := NOT (TP_0.Q OR RS_0.Q1);

END_PROGRAM

// Device/Application/Logic/4.Device/DEVICE_XV1321
PROGRAM DEVICE_XV1321
VAR
	XV1321: BWTS.DEVICE;
END_VAR
VAR // added by the converter: edge detectors and wires of the graphical bodies
    _w1, _w2, _w3 : ANY;
END_VAR

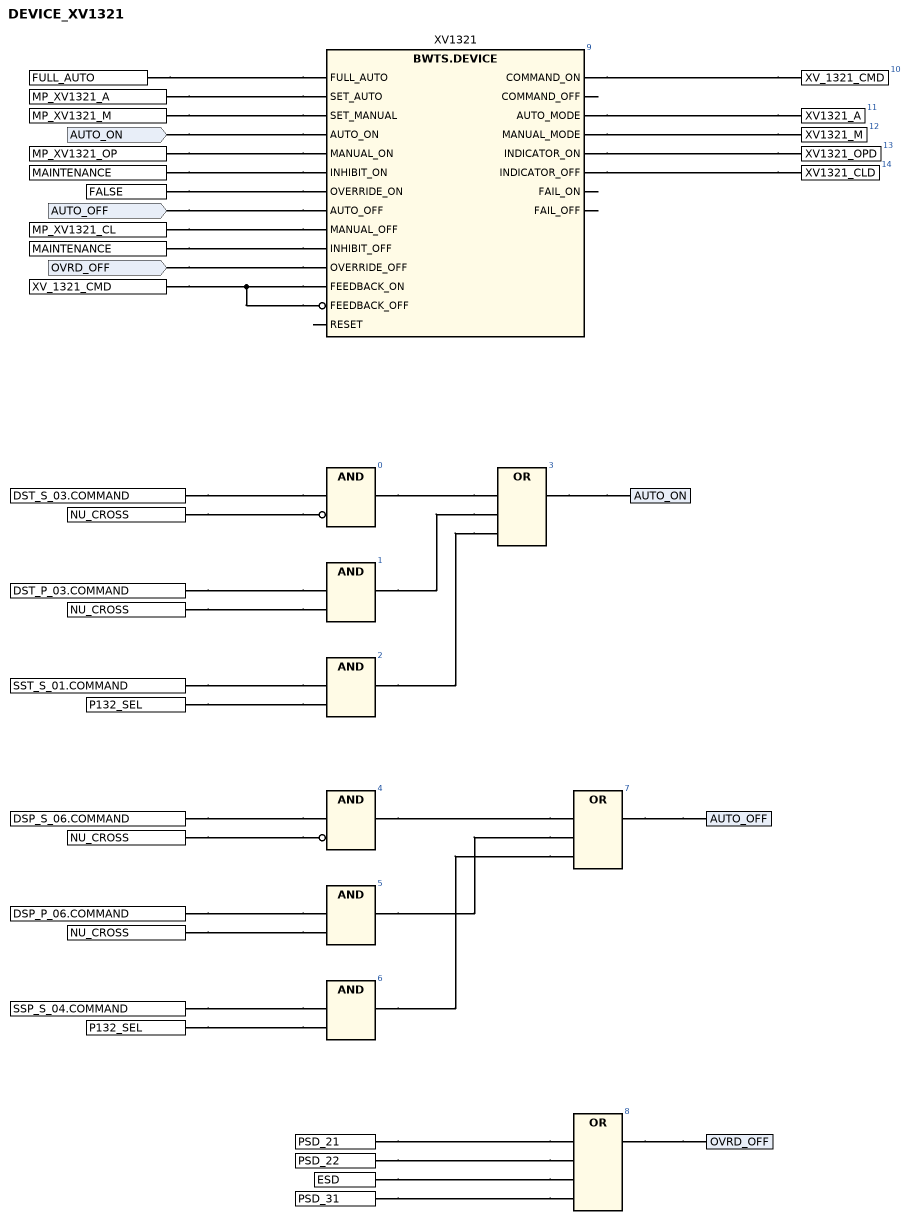
(* DST_S_03.COMMAND AND NOT NU_CROSS OR DST_P_03.COMMAND AND NU_CROSS OR SST_S_01.COMMAND AND P132_SEL; result not used *)
(* DSP_S_06.COMMAND AND NOT NU_CROSS OR DSP_P_06.COMMAND AND NU_CROSS OR SSP_S_04.COMMAND AND P132_SEL; result not used *)
(* PSD_21 OR PSD_22 OR ESD OR PSD_31; result not used *)
XV1321(
    FULL_AUTO := FULL_AUTO,
    SET_AUTO := MP_XV1321_A,
    SET_MANUAL := MP_XV1321_M,
    AUTO_ON := _w1,
    MANUAL_ON := MP_XV1321_OP,
    INHIBIT_ON := MAINTENANCE,
    OVERRIDE_ON := FALSE,
    AUTO_OFF := _w2,
    MANUAL_OFF := MP_XV1321_CL,
    INHIBIT_OFF := MAINTENANCE,
    OVERRIDE_OFF := _w3,
    FEEDBACK_ON := XV_1321_CMD,
    FEEDBACK_OFF := NOT XV_1321_CMD); // BWTS.DEVICE
XV_1321_CMD := XV1321.COMMAND_ON;
XV1321_A := XV1321.AUTO_MODE;
XV1321_M := XV1321.MANUAL_MODE;
XV1321_OPD := XV1321.INDICATOR_ON;
XV1321_CLD := XV1321.INDICATOR_OFF;

END_PROGRAM

// Device/Application/Logic/4.Device/DEVICE_XV2321
PROGRAM DEVICE_XV2321
VAR
	XV2321: BWTS.DEVICE;
END_VAR
VAR // added by the converter: edge detectors and wires of the graphical bodies
    _w1, _w2, _w3 : ANY;
END_VAR

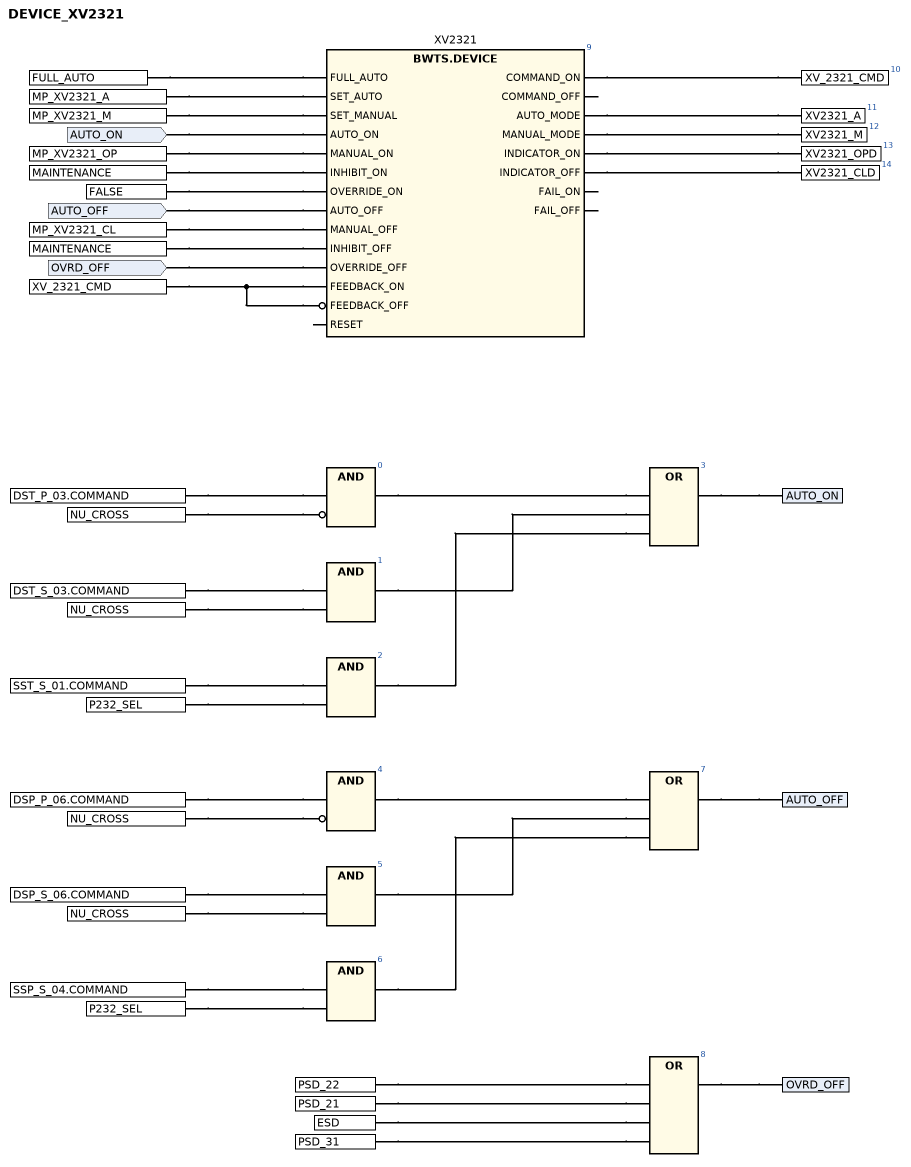
(* DST_P_03.COMMAND AND NOT NU_CROSS OR DST_S_03.COMMAND AND NU_CROSS OR SST_S_01.COMMAND AND P232_SEL; result not used *)
(* DSP_P_06.COMMAND AND NOT NU_CROSS OR DSP_S_06.COMMAND AND NU_CROSS OR SSP_S_04.COMMAND AND P232_SEL; result not used *)
(* PSD_22 OR PSD_21 OR ESD OR PSD_31; result not used *)
XV2321(
    FULL_AUTO := FULL_AUTO,
    SET_AUTO := MP_XV2321_A,
    SET_MANUAL := MP_XV2321_M,
    AUTO_ON := _w1,
    MANUAL_ON := MP_XV2321_OP,
    INHIBIT_ON := MAINTENANCE,
    OVERRIDE_ON := FALSE,
    AUTO_OFF := _w2,
    MANUAL_OFF := MP_XV2321_CL,
    INHIBIT_OFF := MAINTENANCE,
    OVERRIDE_OFF := _w3,
    FEEDBACK_ON := XV_2321_CMD,
    FEEDBACK_OFF := NOT XV_2321_CMD); // BWTS.DEVICE
XV_2321_CMD := XV2321.COMMAND_ON;
XV2321_A := XV2321.AUTO_MODE;
XV2321_M := XV2321.MANUAL_MODE;
XV2321_OPD := XV2321.INDICATOR_ON;
XV2321_CLD := XV2321.INDICATOR_OFF;

END_PROGRAM

// Device/Application/Logic/4.Device/DEVICE_XV1511
PROGRAM DEVICE_XV1511
VAR
	XV1511: BWTS.DEVICE;
END_VAR
VAR // added by the converter: edge detectors and wires of the graphical bodies
    _w1, _w2, _w3, _w4, _w5 : BOOL;
    _w6, _w7, _w8 : ANY;
END_VAR

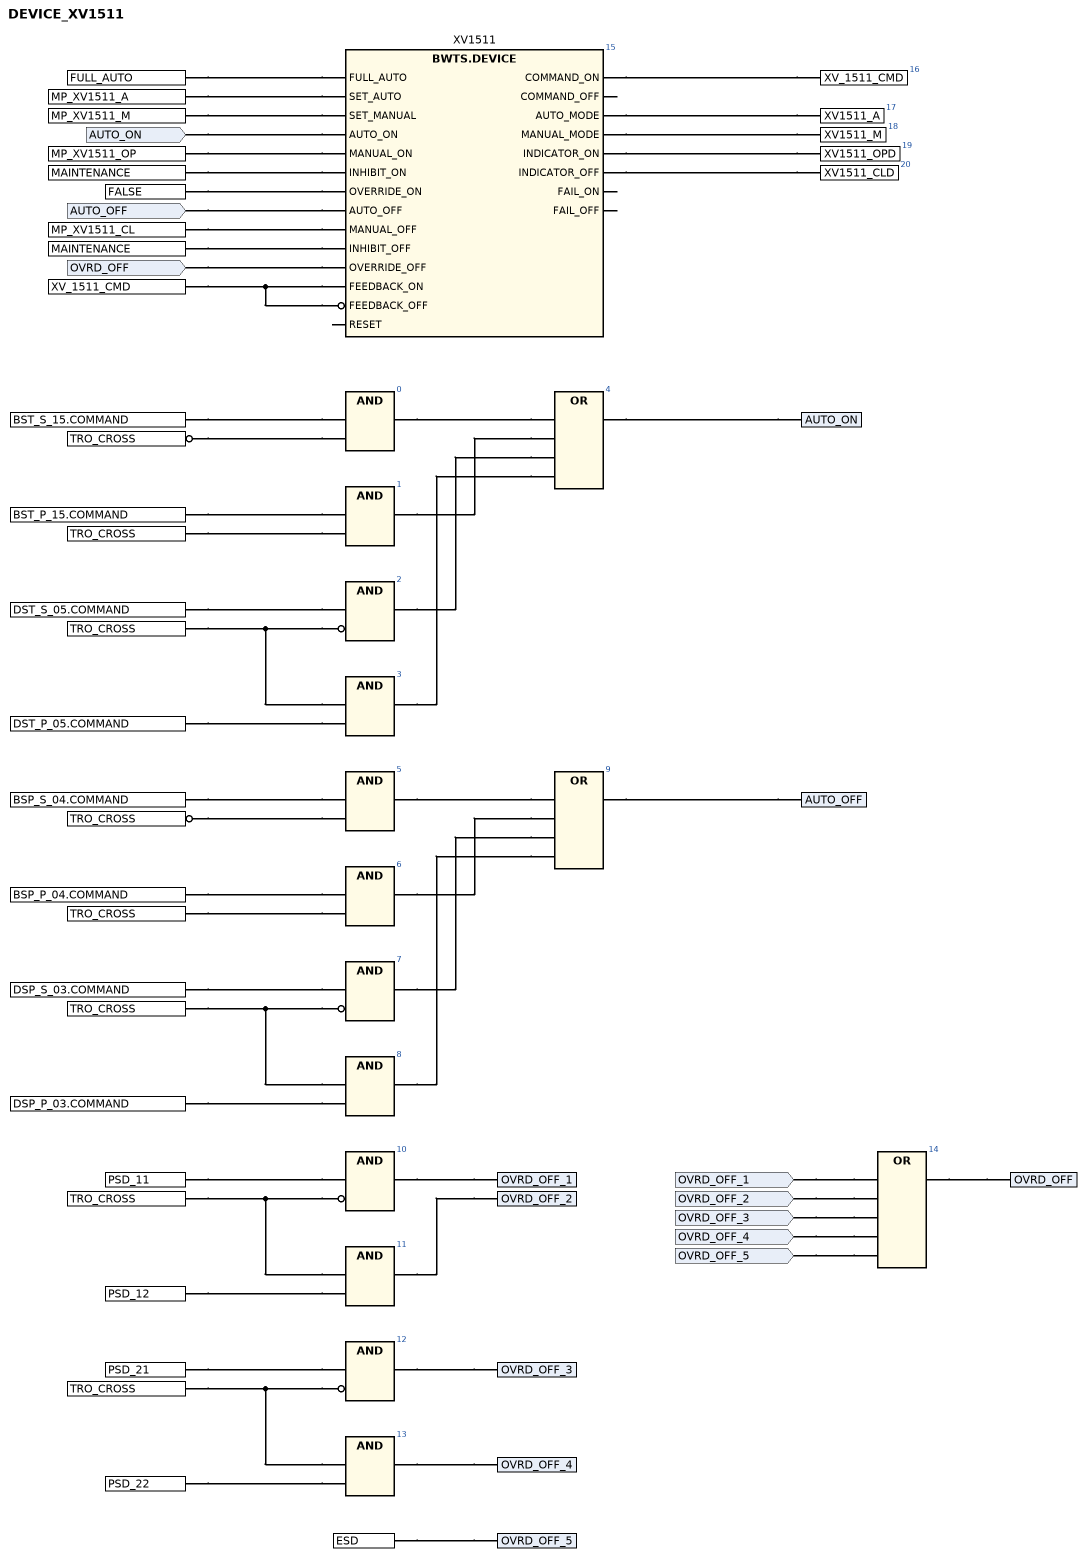
(* BST_S_15.COMMAND AND NOT TRO_CROSS OR BST_P_15.COMMAND AND TRO_CROSS OR DST_S_05.COMMAND AND NOT TRO_CROSS OR TRO_CROSS AND DST_P_05.COMMAND; result not used *)
(* BSP_S_04.COMMAND AND NOT TRO_CROSS OR BSP_P_04.COMMAND AND TRO_CROSS OR DSP_S_03.COMMAND AND NOT TRO_CROSS OR TRO_CROSS AND DSP_P_03.COMMAND; result not used *)
(* PSD_11 AND NOT TRO_CROSS; result not used *)
(* TRO_CROSS AND PSD_12; result not used *)
(* PSD_21 AND NOT TRO_CROSS; result not used *)
(* TRO_CROSS AND PSD_22; result not used *)
(* _w1 OR _w2 OR _w3 OR _w4 OR _w5; result not used *)
XV1511(
    FULL_AUTO := FULL_AUTO,
    SET_AUTO := MP_XV1511_A,
    SET_MANUAL := MP_XV1511_M,
    AUTO_ON := _w6,
    MANUAL_ON := MP_XV1511_OP,
    INHIBIT_ON := MAINTENANCE,
    OVERRIDE_ON := FALSE,
    AUTO_OFF := _w7,
    MANUAL_OFF := MP_XV1511_CL,
    INHIBIT_OFF := MAINTENANCE,
    OVERRIDE_OFF := _w8,
    FEEDBACK_ON := XV_1511_CMD,
    FEEDBACK_OFF := NOT XV_1511_CMD); // BWTS.DEVICE
XV_1511_CMD := XV1511.COMMAND_ON;
XV1511_A := XV1511.AUTO_MODE;
XV1511_M := XV1511.MANUAL_MODE;
XV1511_OPD := XV1511.INDICATOR_ON;
XV1511_CLD := XV1511.INDICATOR_OFF;

END_PROGRAM

// Device/Application/Logic/4.Device/DEVICE_XV1512
PROGRAM DEVICE_XV1512
VAR
	XV1512: BWTS.DEVICE;
END_VAR
VAR // added by the converter: edge detectors and wires of the graphical bodies
    _w1, _w2 : BOOL;
    _w3, _w4, _w5 : ANY;
END_VAR

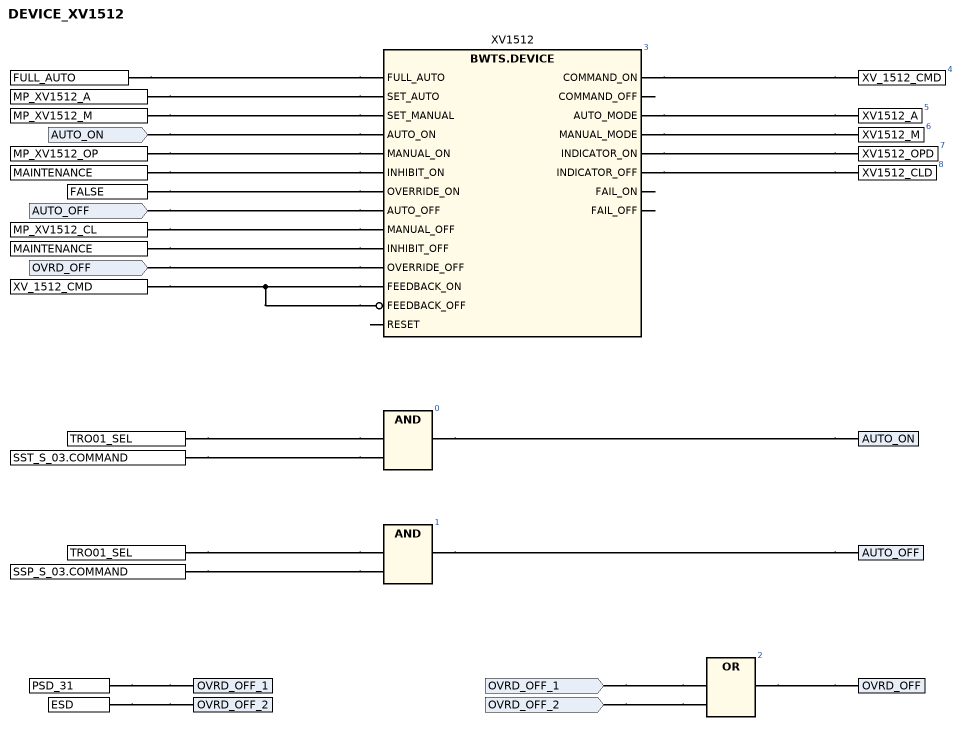
(* TRO01_SEL AND SST_S_03.COMMAND; result not used *)
(* TRO01_SEL AND SSP_S_03.COMMAND; result not used *)
(* _w1 OR _w2; result not used *)
XV1512(
    FULL_AUTO := FULL_AUTO,
    SET_AUTO := MP_XV1512_A,
    SET_MANUAL := MP_XV1512_M,
    AUTO_ON := _w3,
    MANUAL_ON := MP_XV1512_OP,
    INHIBIT_ON := MAINTENANCE,
    OVERRIDE_ON := FALSE,
    AUTO_OFF := _w4,
    MANUAL_OFF := MP_XV1512_CL,
    INHIBIT_OFF := MAINTENANCE,
    OVERRIDE_OFF := _w5,
    FEEDBACK_ON := XV_1512_CMD,
    FEEDBACK_OFF := NOT XV_1512_CMD); // BWTS.DEVICE
XV_1512_CMD := XV1512.COMMAND_ON;
XV1512_A := XV1512.AUTO_MODE;
XV1512_M := XV1512.MANUAL_MODE;
XV1512_OPD := XV1512.INDICATOR_ON;
XV1512_CLD := XV1512.INDICATOR_OFF;

END_PROGRAM

// Device/Application/Logic/4.Device/DEVICE_XV2511
PROGRAM DEVICE_XV2511
VAR
	XV2511: BWTS.DEVICE;
END_VAR
VAR // added by the converter: edge detectors and wires of the graphical bodies
    _w1, _w2, _w3, _w4, _w5 : BOOL;
    _w6, _w7, _w8 : ANY;
END_VAR

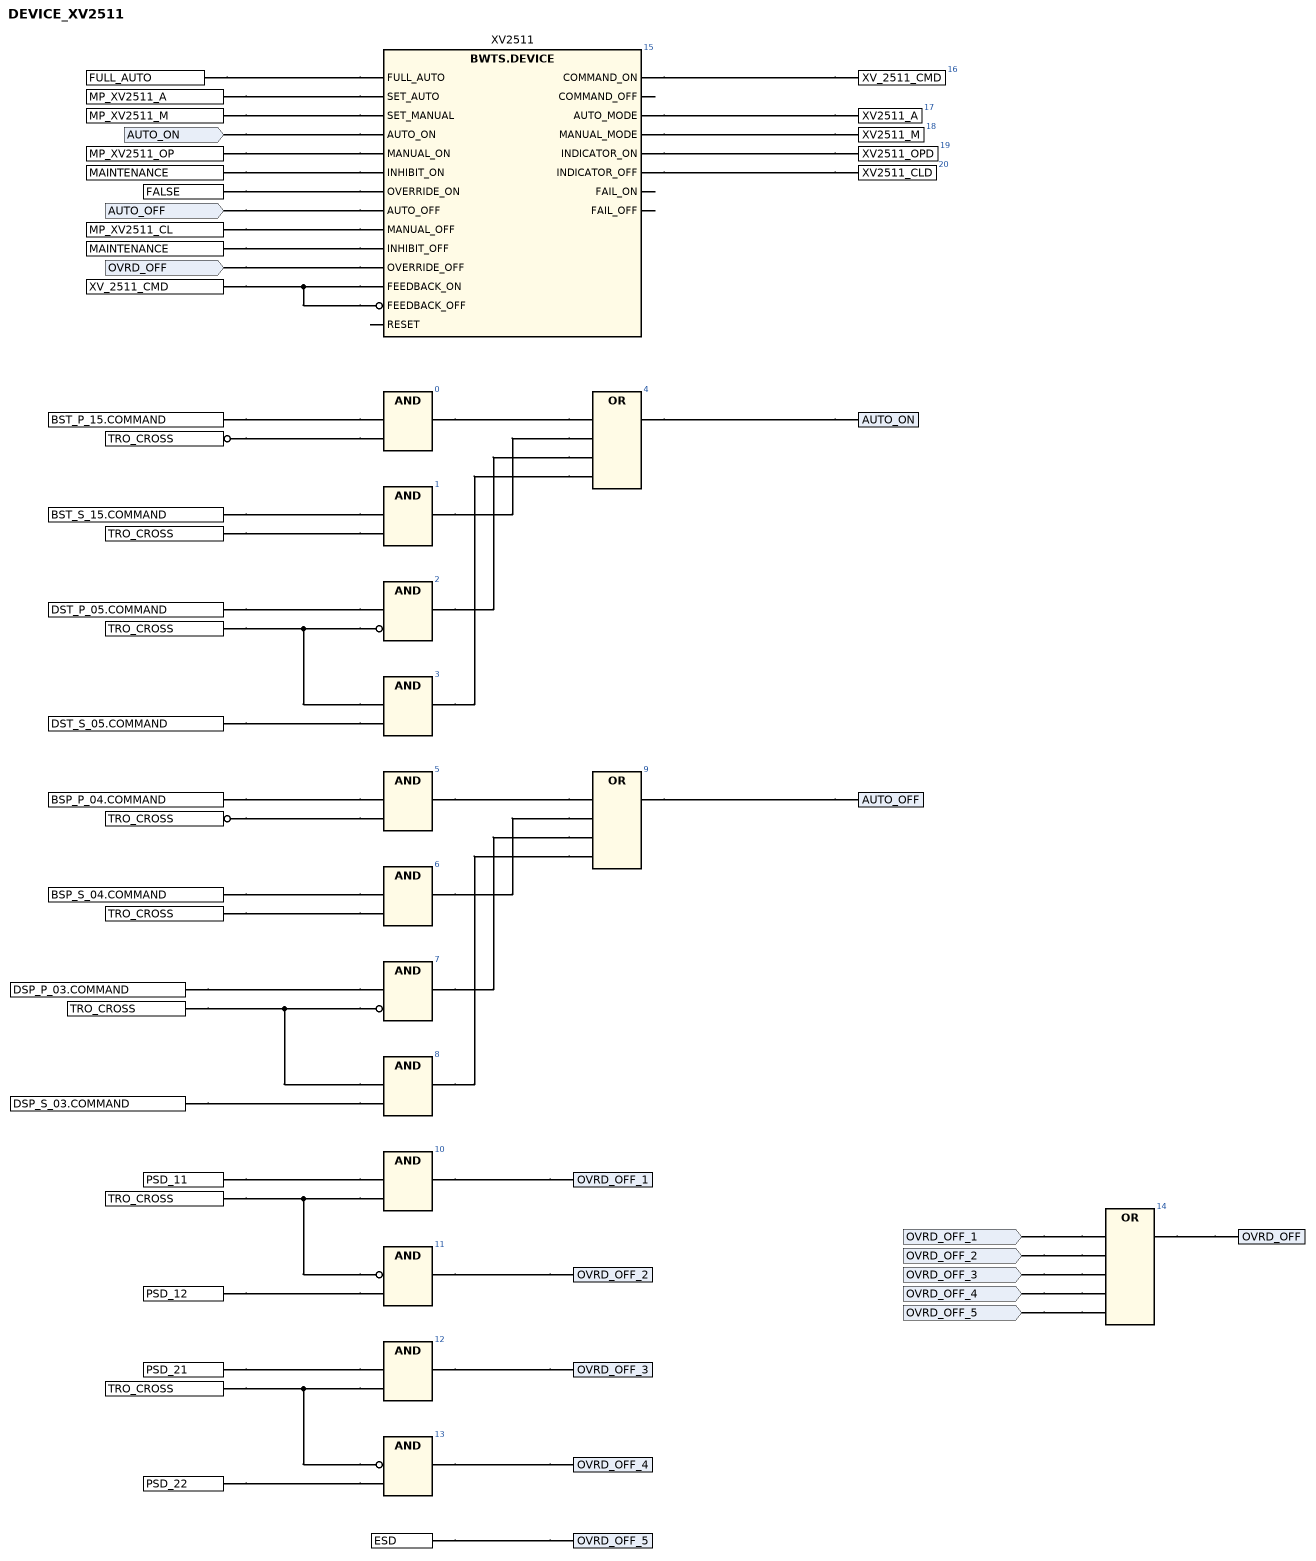
(* BST_P_15.COMMAND AND NOT TRO_CROSS OR BST_S_15.COMMAND AND TRO_CROSS OR DST_P_05.COMMAND AND NOT TRO_CROSS OR TRO_CROSS AND DST_S_05.COMMAND; result not used *)
(* BSP_P_04.COMMAND AND NOT TRO_CROSS OR BSP_S_04.COMMAND AND TRO_CROSS OR DSP_P_03.COMMAND AND NOT TRO_CROSS OR TRO_CROSS AND DSP_S_03.COMMAND; result not used *)
(* PSD_11 AND TRO_CROSS; result not used *)
(* NOT TRO_CROSS AND PSD_12; result not used *)
(* PSD_21 AND TRO_CROSS; result not used *)
(* NOT TRO_CROSS AND PSD_22; result not used *)
(* _w1 OR _w2 OR _w3 OR _w4 OR _w5; result not used *)
XV2511(
    FULL_AUTO := FULL_AUTO,
    SET_AUTO := MP_XV2511_A,
    SET_MANUAL := MP_XV2511_M,
    AUTO_ON := _w6,
    MANUAL_ON := MP_XV2511_OP,
    INHIBIT_ON := MAINTENANCE,
    OVERRIDE_ON := FALSE,
    AUTO_OFF := _w7,
    MANUAL_OFF := MP_XV2511_CL,
    INHIBIT_OFF := MAINTENANCE,
    OVERRIDE_OFF := _w8,
    FEEDBACK_ON := XV_2511_CMD,
    FEEDBACK_OFF := NOT XV_2511_CMD); // BWTS.DEVICE
XV_2511_CMD := XV2511.COMMAND_ON;
XV2511_A := XV2511.AUTO_MODE;
XV2511_M := XV2511.MANUAL_MODE;
XV2511_OPD := XV2511.INDICATOR_ON;
XV2511_CLD := XV2511.INDICATOR_OFF;

END_PROGRAM

// Device/Application/Logic/4.Device/DEVICE_XV2512
PROGRAM DEVICE_XV2512
VAR
	XV2512: BWTS.DEVICE;
END_VAR
VAR // added by the converter: edge detectors and wires of the graphical bodies
    _w1, _w2 : BOOL;
    _w3, _w4, _w5 : ANY;
END_VAR

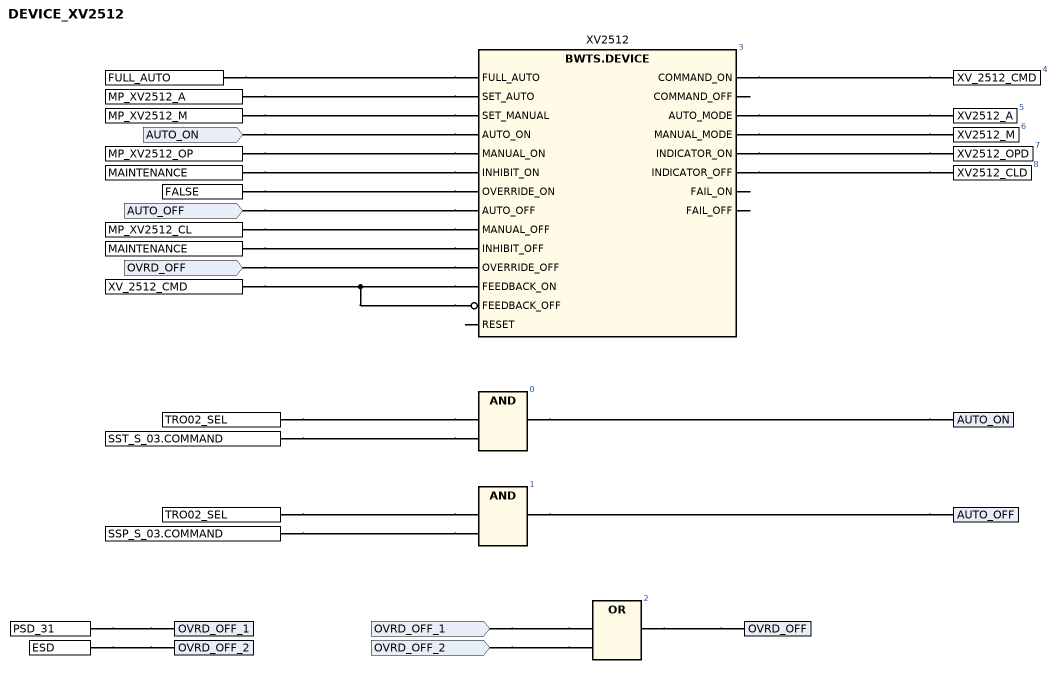
(* TRO02_SEL AND SST_S_03.COMMAND; result not used *)
(* TRO02_SEL AND SSP_S_03.COMMAND; result not used *)
(* _w1 OR _w2; result not used *)
XV2512(
    FULL_AUTO := FULL_AUTO,
    SET_AUTO := MP_XV2512_A,
    SET_MANUAL := MP_XV2512_M,
    AUTO_ON := _w3,
    MANUAL_ON := MP_XV2512_OP,
    INHIBIT_ON := MAINTENANCE,
    OVERRIDE_ON := FALSE,
    AUTO_OFF := _w4,
    MANUAL_OFF := MP_XV2512_CL,
    INHIBIT_OFF := MAINTENANCE,
    OVERRIDE_OFF := _w5,
    FEEDBACK_ON := XV_2512_CMD,
    FEEDBACK_OFF := NOT XV_2512_CMD); // BWTS.DEVICE
XV_2512_CMD := XV2512.COMMAND_ON;
XV2512_A := XV2512.AUTO_MODE;
XV2512_M := XV2512.MANUAL_MODE;
XV2512_OPD := XV2512.INDICATOR_ON;
XV2512_CLD := XV2512.INDICATOR_OFF;

END_PROGRAM

// Device/Application/Logic/4.Device/DEVICE_XV1731
PROGRAM DEVICE_XV1731
VAR
	XV1731: BWTS.DEVICE;
END_VAR
VAR // added by the converter: edge detectors and wires of the graphical bodies
    _w1, _w2, _w3 : ANY;
END_VAR

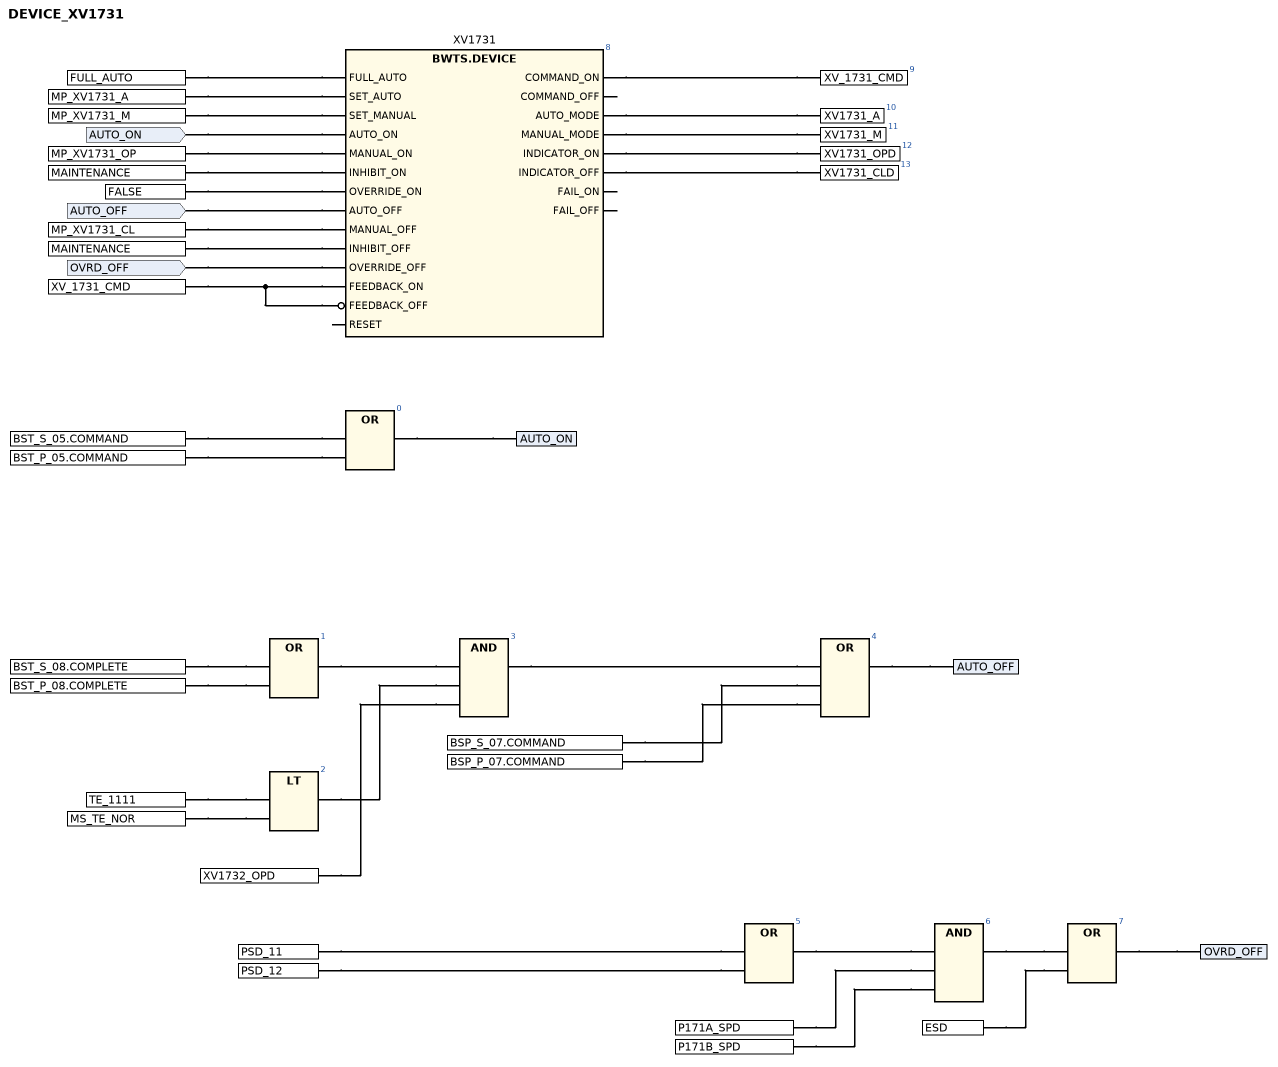
(* BST_S_05.COMMAND OR BST_P_05.COMMAND; result not used *)
(* (BST_S_08.COMPLETE OR BST_P_08.COMPLETE) AND TE_1111 < MS_TE_NOR AND XV1732_OPD OR BSP_S_07.COMMAND OR BSP_P_07.COMMAND; result not used *)
(* (PSD_11 OR PSD_12) AND P171A_SPD AND P171B_SPD OR ESD; result not used *)
XV1731(
    FULL_AUTO := FULL_AUTO,
    SET_AUTO := MP_XV1731_A,
    SET_MANUAL := MP_XV1731_M,
    AUTO_ON := _w1,
    MANUAL_ON := MP_XV1731_OP,
    INHIBIT_ON := MAINTENANCE,
    OVERRIDE_ON := FALSE,
    AUTO_OFF := _w2,
    MANUAL_OFF := MP_XV1731_CL,
    INHIBIT_OFF := MAINTENANCE,
    OVERRIDE_OFF := _w3,
    FEEDBACK_ON := XV_1731_CMD,
    FEEDBACK_OFF := NOT XV_1731_CMD); // BWTS.DEVICE
XV_1731_CMD := XV1731.COMMAND_ON;
XV1731_A := XV1731.AUTO_MODE;
XV1731_M := XV1731.MANUAL_MODE;
XV1731_OPD := XV1731.INDICATOR_ON;
XV1731_CLD := XV1731.INDICATOR_OFF;

END_PROGRAM

// Device/Application/Logic/4.Device/DEVICE_XV1732
PROGRAM DEVICE_XV1732
VAR
	XV1732: BWTS.DEVICE;
END_VAR
VAR // added by the converter: edge detectors and wires of the graphical bodies
    _w1, _w2, _w3 : ANY;
END_VAR

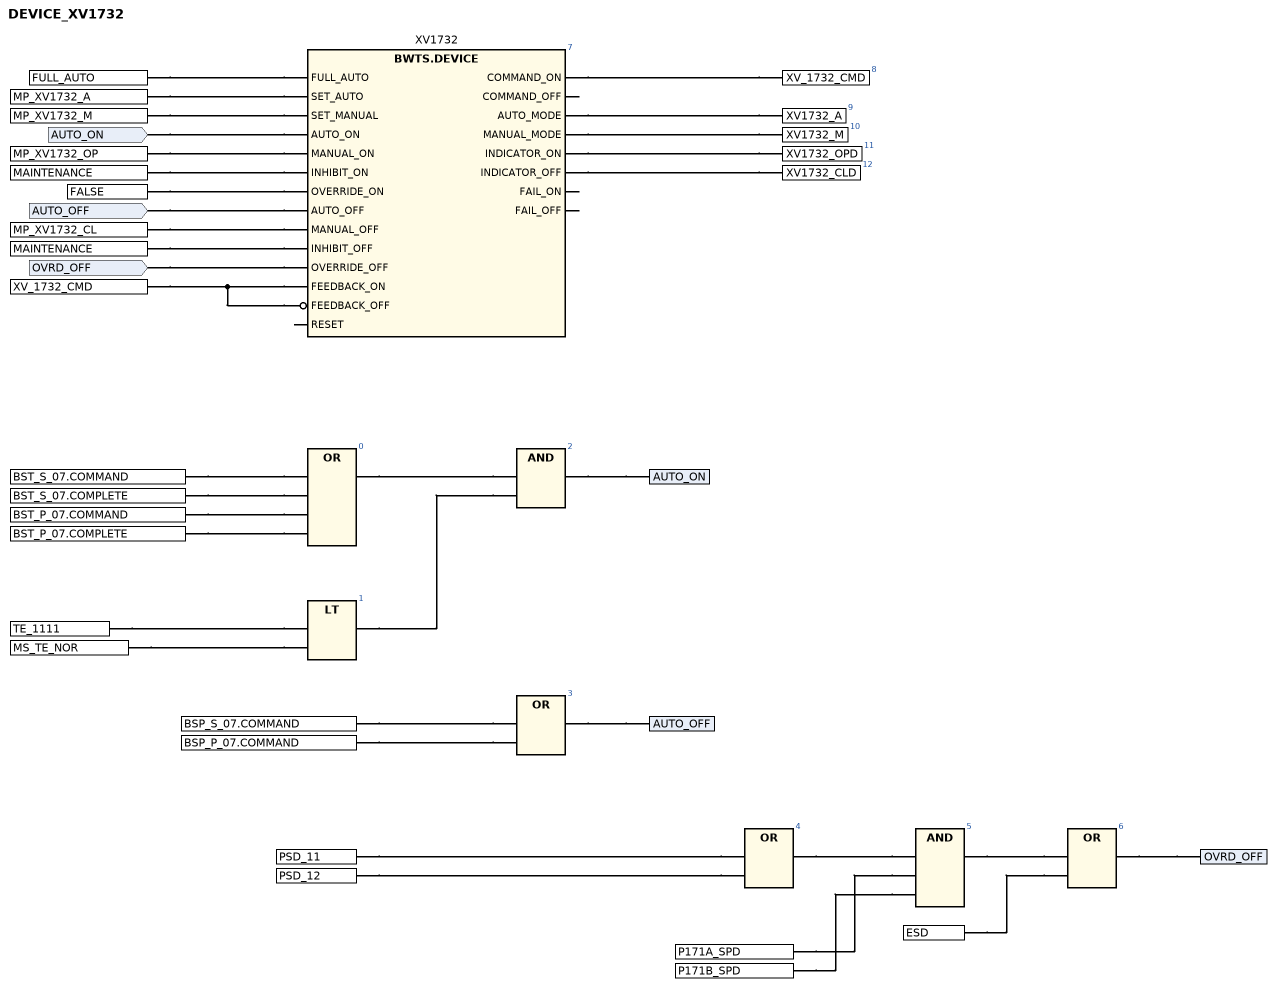
(* (BST_S_07.COMMAND OR BST_S_07.COMPLETE OR BST_P_07.COMMAND OR BST_P_07.COMPLETE) AND TE_1111 < MS_TE_NOR; result not used *)
(* BSP_S_07.COMMAND OR BSP_P_07.COMMAND; result not used *)
(* (PSD_11 OR PSD_12) AND P171A_SPD AND P171B_SPD OR ESD; result not used *)
XV1732(
    FULL_AUTO := FULL_AUTO,
    SET_AUTO := MP_XV1732_A,
    SET_MANUAL := MP_XV1732_M,
    AUTO_ON := _w1,
    MANUAL_ON := MP_XV1732_OP,
    INHIBIT_ON := MAINTENANCE,
    OVERRIDE_ON := FALSE,
    AUTO_OFF := _w2,
    MANUAL_OFF := MP_XV1732_CL,
    INHIBIT_OFF := MAINTENANCE,
    OVERRIDE_OFF := _w3,
    FEEDBACK_ON := XV_1732_CMD,
    FEEDBACK_OFF := NOT XV_1732_CMD); // BWTS.DEVICE
XV_1732_CMD := XV1732.COMMAND_ON;
XV1732_A := XV1732.AUTO_MODE;
XV1732_M := XV1732.MANUAL_MODE;
XV1732_OPD := XV1732.INDICATOR_ON;
XV1732_CLD := XV1732.INDICATOR_OFF;

END_PROGRAM

// Device/Application/Logic/4.Device/DEVICE_XV1901
PROGRAM DEVICE_XV1901
VAR
	XV1901 : BWTS.DEVICE;
END_VAR
VAR // added by the converter: edge detectors and wires of the graphical bodies
    _w1, _w2, _w3 : ANY;
END_VAR

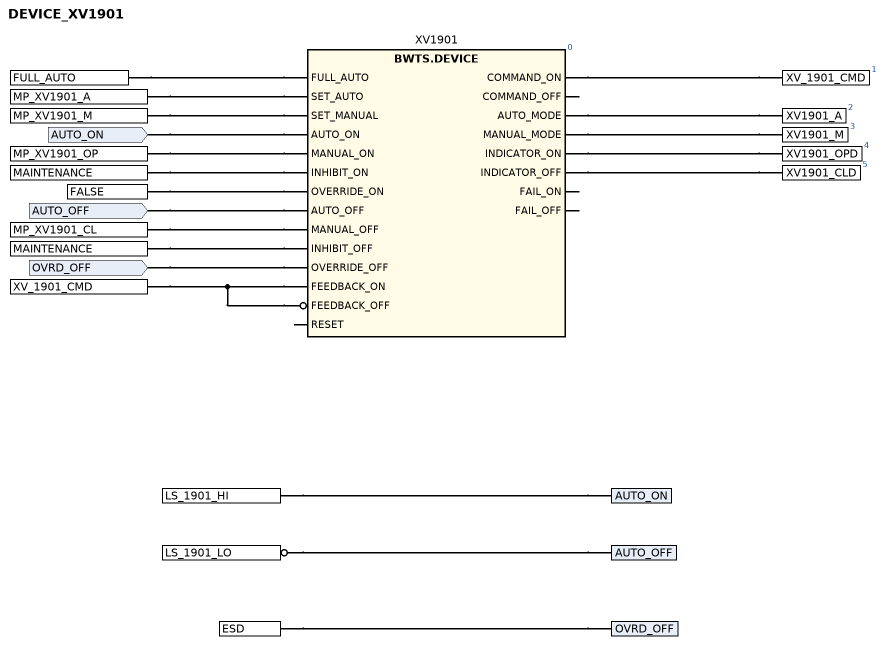
XV1901(
    FULL_AUTO := FULL_AUTO,
    SET_AUTO := MP_XV1901_A,
    SET_MANUAL := MP_XV1901_M,
    AUTO_ON := _w1,
    MANUAL_ON := MP_XV1901_OP,
    INHIBIT_ON := MAINTENANCE,
    OVERRIDE_ON := FALSE,
    AUTO_OFF := _w2,
    MANUAL_OFF := MP_XV1901_CL,
    INHIBIT_OFF := MAINTENANCE,
    OVERRIDE_OFF := _w3,
    FEEDBACK_ON := XV_1901_CMD,
    FEEDBACK_OFF := NOT XV_1901_CMD); // BWTS.DEVICE
XV_1901_CMD := XV1901.COMMAND_ON;
XV1901_A := XV1901.AUTO_MODE;
XV1901_M := XV1901.MANUAL_MODE;
XV1901_OPD := XV1901.INDICATOR_ON;
XV1901_CLD := XV1901.INDICATOR_OFF;

END_PROGRAM

// Device/Application/Logic/4.Device/DEVICE_XV1541
PROGRAM DEVICE_XV1541
VAR
	XV1541: BWTS.DEVICE;
END_VAR
VAR // added by the converter: edge detectors and wires of the graphical bodies
    _w1, _w2, _w3 : ANY;
END_VAR

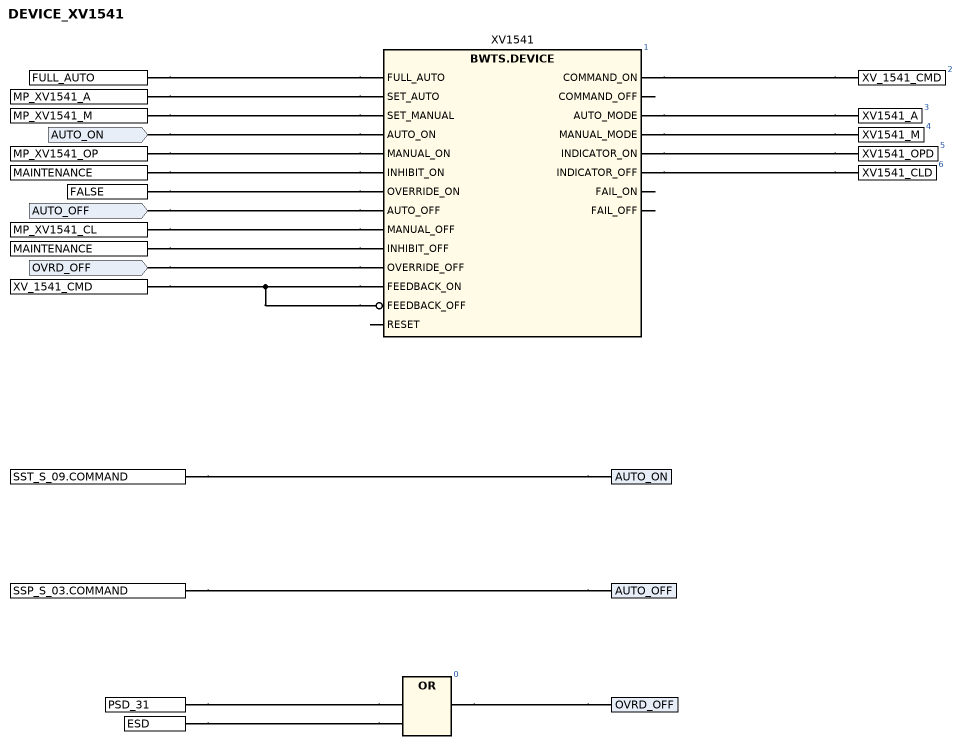
(* PSD_31 OR ESD; result not used *)
XV1541(
    FULL_AUTO := FULL_AUTO,
    SET_AUTO := MP_XV1541_A,
    SET_MANUAL := MP_XV1541_M,
    AUTO_ON := _w1,
    MANUAL_ON := MP_XV1541_OP,
    INHIBIT_ON := MAINTENANCE,
    OVERRIDE_ON := FALSE,
    AUTO_OFF := _w2,
    MANUAL_OFF := MP_XV1541_CL,
    INHIBIT_OFF := MAINTENANCE,
    OVERRIDE_OFF := _w3,
    FEEDBACK_ON := XV_1541_CMD,
    FEEDBACK_OFF := NOT XV_1541_CMD); // BWTS.DEVICE
XV_1541_CMD := XV1541.COMMAND_ON;
XV1541_A := XV1541.AUTO_MODE;
XV1541_M := XV1541.MANUAL_MODE;
XV1541_OPD := XV1541.INDICATOR_ON;
XV1541_CLD := XV1541.INDICATOR_OFF;

END_PROGRAM

// Device/Application/Logic/3.SD/ESD101
PROGRAM ESD101
VAR
	RS_0: RS;
	TP_0: TP;
END_VAR

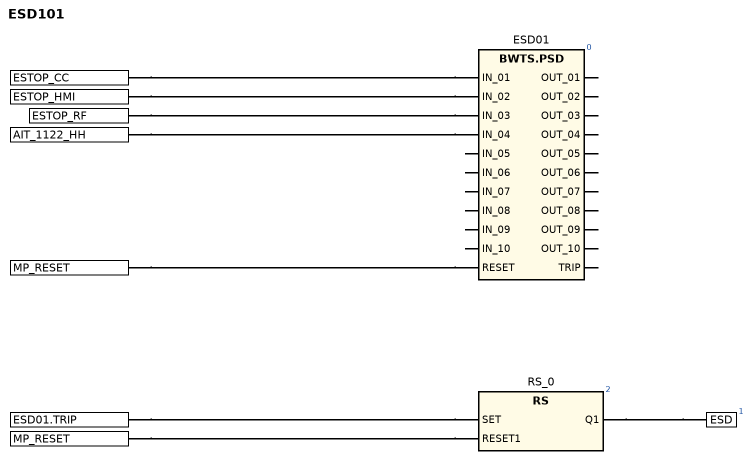
ESD01(IN_01 := ESTOP_CC, IN_02 := ESTOP_HMI, IN_03 := ESTOP_RF, IN_04 := AIT_1122_HH, RESET := MP_RESET); // BWTS.PSD
ESD := RS_0.Q1;
RS_0(SET := ESD01.TRIP, RESET1 := MP_RESET); // RS

END_PROGRAM

// Device/Application/Logic/3.SD/PSD10X
PROGRAM PSD10X
VAR
	TON_0: TON;
END_VAR
VAR // added by the converter: edge detectors and wires of the graphical bodies
    _w1, _w2, _w3, _w4, _w5, _w8, _w9, _w10, _w11, _w12, _w13, _w14, _w15, _w16, _w17 : ANY;
    _w6, _w7 : BOOL;
END_VAR

